KUKA KRL program: MyProgram_113().src

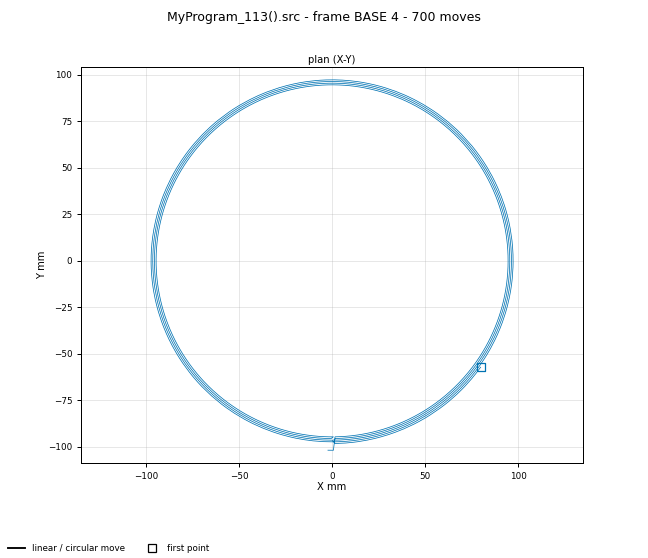
[picture p0: tool path of MyProgram_113().src in frame BASE 4, 700 of 700 moves have a stored position in this frame; points joined in program order, loops and branches not executed]
&ACCESS RVP
&REL 1
&PARAM TEMPLATE = C:\KRC\Roboter\Template\vorgabe
&PARAM EDITMASK = *
DEF MyProgram_113()
; ---- Setting reference (Base) ----
$BASE = BASE_DATA[4]

; --------------------------
; ---- Setting tool (TCP) ----
$TOOL = TOOL_DATA[3]
; --------------------------

$VEL.CP = VEL_APROX_PRINT
Startdeposition()
$VEL.CP = VEL_PRINT
LIN {X 79.7976,Y -57.1488,Z 98,A -40.8571,B 24.9367,C -1.8375,E1 25.1286,E2 126.2832} C_DIS
LIN {X 77.2204,Y -60.5867,Z 98,A -43.0229,B 24.9363,C -1.844,E1 25.125,E2 128.4234} C_DIS
LIN {X 74.8763,Y -63.4603,Z 98,A -45.4458,B 24.9373,C -1.8284,E1 25.1206,E2 130.8721} C_DIS
LIN {X 71.3027,Y -67.4509,Z 98,A -48.1343,B 24.9367,C -1.8374,E1 25.1156,E2 133.5274} C_DIS
LIN {X 69.3871,Y -69.4217,Z 98,A -49.9709,B 24.9376,C -1.8245,E1 25.1119,E2 135.3867} C_DIS
LIN {X 66.9172,Y -71.8046,Z 98,A -52.0394,B 24.9381,C -1.8172,E1 25.1077,E2 137.4638} C_DIS
LIN {X 62.9842,Y -75.2776,Z 98,A -54.7785,B 24.9377,C -1.8227,E1 25.102,E2 140.1792} C_DIS
LIN {X 60.5437,Y -77.2543,Z 98,A -56.7758,B 24.9384,C -1.8124,E1 25.0976,E2 142.1934} C_DIS
LIN {X 58.0242,Y -79.1632,Z 98,A -58.7964,B 24.9391,C -1.8018,E1 25.093,E2 144.2318} C_DIS
LIN {X 52.4588,Y -82.9577,Z 98,A -62.2953,B 24.9386,C -1.8106,E1 25.085,E2 147.6983} C_DIS
LIN {X 50.2118,Y -84.3355,Z 98,A -64.0193,B 24.9392,C -1.8007,E1 25.0808,E2 149.4404} C_DIS
LIN {X 46.9316,Y -86.2036,Z 98,A -66.5927,B 24.9404,C -1.7828,E1 25.0744,E2 152.0485} C_DIS
LIN {X 44.0309,Y -87.7219,Z 98,A -68.1285,B 24.9397,C -1.7938,E1 25.0707,E2 153.5542} C_DIS
LIN {X 38.5072,Y -90.2828,Z 98,A -71.4077,B 24.9394,C -1.7987,E1 25.0624,E2 156.8136} C_DIS
LIN {X 33.9539,Y -92.0916,Z 98,A -74.5314,B 24.9403,C -1.7848,E1 25.0542,E2 159.9633} C_DIS
LIN {X 30.3745,Y -93.3329,Z 98,A -76.7207,B 24.9404,C -1.7828,E1 25.0484,E2 162.1529} C_DIS
LIN {X 26.2417,Y -94.5794,Z 98,A -79.2585,B 24.9407,C -1.7793,E1 25.0416,E2 164.6947} C_DIS
LIN {X 22.9791,Y -95.4236,Z 98,A -81.814,B 24.9422,C -1.7557,E1 25.0345,E2 167.3025} C_DIS
LIN {X 18.9563,Y -96.3039,Z 98,A -83.7662,B 24.9413,C -1.7702,E1 25.0293,E2 169.218} C_DIS
LIN {X 13.978,Y -97.1507,Z 98,A -86.15,B 24.94,C -1.7888,E1 25.0228,E2 171.5551} C_DIS
LIN {X 11.5893,Y -97.4645,Z 98,A -88.6482,B 24.9427,C -1.7479,E1 25.0156,E2 174.1484} C_DIS
LIN {X 7.1702,Y -97.8893,Z 98,A -90.2748,B 24.9405,C -1.7818,E1 25.0113,E2 175.6938} C_DIS
LIN {X 1.7256,Y -98.1358,Z 98,A -93.4363,B 24.9405,C -1.7814,E1 25.0025,E2 178.8555} C_DIS
LIN {X 1.7256,Y -98.1358,Z 98,A -93.4363,B 24.9405,C -1.7814,E1 25.0025,E2 178.8555} C_DIS
Enddeposition()
LIN {X 0.7021,Y -97.2501,Z 98,A -94.9609,B 24.9417,C -1.7637,E1 24.9981,E2 180.4219} C_DIS
Startdeposition()
$VEL.CP = VEL_PRINT
LIN {X 3.3521,Y -97.1984,Z 98,A -91.5255,B 24.9371,C -1.832,E1 25.0082,E2 176.8251} C_DIS
LIN {X 7.9705,Y -96.9286,Z 98,A -88.6357,B 24.9366,C -1.8394,E1 25.0163,E2 173.9192} C_DIS
LIN {X 11.4013,Y -96.5849,Z 98,A -87.1457,B 24.9379,C -1.8205,E1 25.0203,E2 172.4751} C_DIS
LIN {X 14.7868,Y -96.1248,Z 98,A -85.2922,B 24.9382,C -1.8159,E1 25.0254,E2 170.6339} C_DIS
LIN {X 18.9278,Y -95.3974,Z 98,A -82.0938,B 24.9362,C -1.8449,E1 25.0343,E2 167.3706} C_DIS
LIN {X 22.4173,Y -94.6382,Z 98,A -80.5089,B 24.9374,C -1.8274,E1 25.0385,E2 165.8293} C_DIS
LIN {X 25.8034,Y -93.7711,Z 98,A -78.594,B 24.9376,C -1.8242,E1 25.0436,E2 163.9251} C_DIS
LIN {X 28.6619,Y -92.9362,Z 98,A -76.7124,B 24.9372,C -1.831,E1 25.0487,E2 162.0308} C_DIS
LIN {X 31.9858,Y -91.8454,Z 98,A -74.7403,B 24.9372,C -1.8302,E1 25.0539,E2 160.0644} C_DIS
LIN {X 36.6622,Y -90.0806,Z 98,A -71.8461,B 24.9371,C -1.8323,E1 25.0615,E2 157.1714} C_DIS
LIN {X 38.538,Y -89.2943,Z 98,A -69.8507,B 24.9348,C -1.8645,E1 25.0668,E2 155.1047} C_DIS
LIN {X 42.308,Y -87.5711,Z 98,A -68.0871,B 24.9364,C -1.8424,E1 25.0711,E2 153.398} C_DIS
LIN {X 44.7573,Y -86.3462,Z 98,A -66.3081,B 24.9357,C -1.8514,E1 25.0755,E2 151.6026} C_DIS
LIN {X 51.0632,Y -82.7737,Z 98,A -62.3793,B 24.9361,C -1.846,E1 25.085,E2 147.6983} C_DIS
LIN {X 55.4802,Y -79.8785,Z 98,A -58.6183,B 24.9339,C -1.8772,E1 25.0938,E2 143.8761} C_DIS
LIN {X 58.3576,Y -77.8012,Z 98,A -57.0633,B 24.9351,C -1.8609,E1 25.0972,E2 142.3654} C_DIS
LIN {X 61.0225,Y -75.7295,Z 98,A -55.3486,B 24.9355,C -1.8546,E1 25.1009,E2 140.6718} C_DIS
LIN {X 64.4955,Y -72.7957,Z 98,A -51.9466,B 24.9331,C -1.8888,E1 25.1082,E2 137.2025} C_DIS
LIN {X 66.9498,Y -70.5447,Z 98,A -50.4816,B 24.9342,C -1.8741,E1 25.1111,E2 135.7782} C_DIS
LIN {X 69.097,Y -68.4416,Z 98,A -48.7316,B 24.9339,C -1.8776,E1 25.1146,E2 134.0274} C_DIS
LIN {X 72.4346,Y -64.8989,Z 98,A -45.2556,B 24.9317,C -1.9087,E1 25.1213,E2 130.4932} C_DIS
LIN {X 74.9309,Y -62.0003,Z 98,A -43.6411,B 24.9331,C -1.8894,E1 25.1241,E2 128.9315} C_DIS
LIN {X 76.9346,Y -59.4956,Z 98,A -41.0568,B 24.9308,C -1.9218,E1 25.1286,E2 126.283} C_DIS
LIN {X 79.3962,Y -56.1696,Z 98,A -39.1586,B 24.9318,C -1.9072,E1 25.1316,E2 124.4285} C_DIS
LIN {X 81.8934,Y -52.4605,Z 98,A -36.5864,B 24.9315,C -1.9122,E1 25.1355,E2 121.8573} C_DIS
LIN {X 83.2034,Y -50.3573,Z 98,A -34.6449,B 24.9298,C -1.9354,E1 25.1384,E2 119.8709} C_DIS
LIN {X 85.1347,Y -47.0204,Z 98,A -33.2212,B 24.9317,C -1.9086,E1 25.1403,E2 118.518} C_DIS
LIN {X 87.4131,Y -42.6369,Z 98,A -29.992,B 24.9302,C -1.9297,E1 25.1444,E2 115.2561} C_DIS
LIN {X 88.8191,Y -39.6224,Z 98,A -28.2174,B 24.9302,C -1.9283,E1 25.1464,E2 113.4944} C_DIS
LIN {X 90.266,Y -36.2067,Z 98,A -25.8677,B 24.9293,C -1.9415,E1 25.149,E2 111.1265} C_DIS
LIN {X 91.5506,Y -32.8238,Z 98,A -23.7356,B 24.9288,C -1.9481,E1 25.151,E2 108.9907} C_DIS
LIN {X 93.2043,Y -27.7776,Z 98,A -20.6688,B 24.9283,C -1.9555,E1 25.1536,E2 105.924} C_DIS
LIN {X 94.208,Y -24.1556,Z 98,A -18.5095,B 24.9279,C -1.9603,E1 25.1552,E2 103.7657} C_DIS
LIN {X 95.2371,Y -19.7115,Z 98,A -16.2285,B 24.9285,C -1.9529,E1 25.1566,E2 101.5155} C_DIS
LIN {X 95.9344,Y -15.9756,Z 98,A -13.6784,B 24.9271,C -1.9723,E1 25.1578,E2 98.9345} C_DIS
LIN {X 96.4194,Y -12.7275,Z 98,A -11.7354,B 24.9266,C -1.9788,E1 25.1586,E2 96.9876} C_DIS
LIN {X 96.7838,Y -9.5822,Z 98,A -9.6481,B 24.9255,C -1.9936,E1 25.1592,E2 94.8777} C_DIS
LIN {X 97.1972,Y -3.3908,Z 98,A -6.1803,B 24.9252,C -1.998,E1 25.1597,E2 91.4203} C_DIS
LIN {X 97.2518,Y -0.8973,Z 98,A -4.0584,B 24.9228,C -2.0287,E1 25.1597,E2 89.2385} C_DIS
LIN {X 97.1951,Y 3.4602,Z 98,A -2.3961,B 24.9249,C -2.0009,E1 25.1597,E2 87.6515} C_DIS
LIN {X 96.9672,Y 7.4872,Z 98,A 0.1195,B 24.9239,C -2.014,E1 25.1592,E2 85.12} C_DIS
LIN {X 96.6458,Y 10.8814,Z 98,A 2.1602,B 24.9234,C -2.0217,E1 25.1586,E2 83.0734} C_DIS
LIN {X 95.684,Y 17.4137,Z 98,A 6.0714,B 24.9224,C -2.0347,E1 25.1569,E2 79.1543} C_DIS
LIN {X 94.9676,Y 20.9723,Z 98,A 8.0982,B 24.9222,C -2.0369,E1 25.1557,E2 77.1341} C_DIS
LIN {X 94.1017,Y 24.5689,Z 98,A 10.2032,B 24.9219,C -2.0407,E1 25.1543,E2 75.0324} C_DIS
LIN {X 93.2925,Y 27.4805,Z 98,A 12.0287,B 24.9214,C -2.0479,E1 25.1529,E2 73.2003} C_DIS
LIN {X 92.4694,Y 30.1344,Z 98,A 14.4718,B 24.9185,C -2.0846,E1 25.1507,E2 70.6845} C_DIS
LIN {X 90.9388,Y 34.4784,Z 98,A 16.3375,B 24.9205,C -2.0592,E1 25.149,E2 68.8892} C_DIS
LIN {X 89.01,Y 39.1915,Z 98,A 19.9629,B 24.9179,C -2.0923,E1 25.145,E2 65.2054} C_DIS
LIN {X 87.3478,Y 42.7693,Z 98,A 21.6868,B 24.9192,C -2.0753,E1 25.1429,E2 63.531} C_DIS
LIN {X 85.9471,Y 45.5167,Z 98,A 24.5151,B 24.9157,C -2.12,E1 25.1391,E2 60.612} C_DIS
LIN {X 83.2177,Y 50.3337,Z 98,A 27.2311,B 24.9167,C -2.1072,E1 25.1352,E2 57.9401} C_DIS
LIN {X 81.3082,Y 53.3634,Z 98,A 29.2555,B 24.9166,C -2.1093,E1 25.1322,E2 55.9209} C_DIS
LIN {X 79.4218,Y 56.1337,Z 98,A 30.8335,B 24.9174,C -2.0988,E1 25.1297,E2 54.3753} C_DIS
LIN {X 77.2022,Y 59.1483,Z 98,A 33.4101,B 24.9158,C -2.1186,E1 25.1253,E2 51.7642} C_DIS
LIN {X 75.1203,Y 61.7724,Z 98,A 35.1259,B 24.9162,C -2.1133,E1 25.1223,E2 50.069} C_DIS
LIN {X 69.4071,Y 68.1276,Z 98,A 39.9538,B 24.916,C -2.1165,E1 25.1132,E2 45.2548} C_DIS
LIN {X 67.1097,Y 70.3932,Z 98,A 42.2478,B 24.9145,C -2.1355,E1 25.1085,E2 42.9253} C_DIS
LIN {X 62.2387,Y 74.7328,Z 98,A 45.8912,B 24.9145,C -2.1354,E1 25.1008,E2 39.2965} C_DIS
LIN {X 56.8744,Y 78.8933,Z 98,A 49.6994,B 24.9145,C -2.1352,E1 25.0924,E2 35.5026} C_DIS
LIN {X 53.8448,Y 80.9908,Z 98,A 52.9079,B 24.911,C -2.1781,E1 25.0847,E2 32.2033} C_DIS
LIN {X 48.9624,Y 84.0336,Z 98,A 55.057,B 24.9144,C -2.1362,E1 25.0798,E2 30.16} C_DIS
LIN {X 44.2162,Y 86.6231,Z 98,A 58.4066,B 24.9136,C -2.1466,E1 25.0715,E2 26.7953} C_DIS
LIN {X 40.9897,Y 88.1956,Z 98,A 60.4692,B 24.9136,C -2.1472,E1 25.0663,E2 24.7366} C_DIS
LIN {X 38.9606,Y 89.1106,Z 98,A 62.7877,B 24.9103,C -2.1862,E1 25.0602,E2 22.3313} C_DIS
LIN {X 33.9331,Y 91.1453,Z 98,A 64.9612,B 24.9132,C -2.1512,E1 25.0547,E2 20.2454} C_DIS
LIN {X 28.6134,Y 92.9513,Z 98,A 68.0623,B 24.9136,C -2.1463,E1 25.0466,E2 17.1619} C_DIS
LIN {X 25.915,Y 93.7406,Z 98,A 69.9785,B 24.9127,C -2.1569,E1 25.0414,E2 15.2237} C_DIS
LIN {X 22.9884,Y 94.4995,Z 98,A 71.6259,B 24.913,C -2.1531,E1 25.0369,E2 13.5878} C_DIS
LIN {X 19.7066,Y 95.2381,Z 98,A 73.6718,B 24.9128,C -2.1564,E1 25.0313,E2 11.5368} C_DIS
LIN {X 16.4675,Y 95.8522,Z 98,A 75.666,B 24.9126,C -2.159,E1 25.0258,E2 9.5386} C_DIS
LIN {X 13.9554,Y 96.2494,Z 98,A 77.9138,B 24.9103,C -2.1866,E1 25.0195,E2 7.2272} C_DIS
LIN {X 9.3981,Y 96.8014,Z 98,A 79.9182,B 24.9124,C -2.1616,E1 25.0141,E2 5.2835} C_DIS
LIN {X 5.6176,Y 97.0934,Z 98,A 81.9493,B 24.9129,C -2.1544,E1 25.0084,E2 3.2704} C_DIS
LIN {X 1.3581,Y 97.247,Z 98,A 84.4198,B 24.9131,C -2.1527,E1 25.0016,E2 0.8045} C_DIS
LIN {X -3.1957,Y 97.2032,Z 98,A 87.2707,B 24.9127,C -2.158,E1 24.9936,E2 -2.0591} C_DIS
LIN {X -6.5423,Y 97.0352,Z 98,A 89.0987,B 24.9131,C -2.1521,E1 24.9885,E2 -3.8736} C_DIS
LIN {X -8.6993,Y 96.8659,Z 98,A 90.8129,B 24.9119,C -2.167,E1 24.9836,E2 -5.6241} C_DIS
LIN {X -14.1209,Y 96.2259,Z 98,A 93.7478,B 24.9129,C -2.1551,E1 24.9756,E2 -8.5328} C_DIS
LIN {X -17.3852,Y 95.6892,Z 98,A 95.5906,B 24.9133,C -2.1499,E1 24.9705,E2 -10.3653} C_DIS
LIN {X -20.594,Y 95.0502,Z 98,A 97.6154,B 24.9132,C -2.1517,E1 24.965,E2 -12.3966} C_DIS
LIN {X -24.4571,Y 94.1305,Z 98,A 100.7061,B 24.9112,C -2.1757,E1 24.9565,E2 -15.5489} C_DIS
LIN {X -28.6765,Y 92.9317,Z 98,A 102.5615,B 24.9135,C -2.1474,E1 24.9517,E2 -17.3401} C_DIS
LIN {X -34.996,Y 90.7419,Z 98,A 106.4035,B 24.9142,C -2.139,E1 24.9416,E2 -21.1696} C_DIS
LIN {X -39.6014,Y 88.8282,Z 98,A 109.857,B 24.9131,C -2.1524,E1 24.9326,E2 -24.6633} C_DIS
LIN {X -44.1812,Y 86.641,Z 98,A 112.429,B 24.9146,C -2.1333,E1 24.9263,E2 -27.1965} C_DIS
LIN {X -50.0589,Y 83.3847,Z 98,A 116.4561,B 24.915,C -2.1286,E1 24.9165,E2 -31.2242} C_DIS
LIN {X -52.8436,Y 81.6475,Z 98,A 118.4417,B 24.9152,C -2.1268,E1 24.9118,E2 -33.2118} C_DIS
LIN {X -55.4064,Y 79.9298,Z 98,A 120.486,B 24.9148,C -2.1308,E1 24.9071,E2 -35.2727} C_DIS
LIN {X -60.9712,Y 75.7711,Z 98,A 124.3317,B 24.9162,C -2.1138,E1 24.8986,E2 -39.0918} C_DIS
LIN {X -62.9622,Y 74.1243,Z 98,A 126.2604,B 24.9154,C -2.1241,E1 24.8944,E2 -41.0525} C_DIS
LIN {X -65.4196,Y 71.966,Z 98,A 127.5675,B 24.9174,C -2.0989,E1 24.8918,E2 -42.3048} C_DIS
LIN {X -69.6493,Y 67.8814,Z 98,A 131.1261,B 24.9178,C -2.0937,E1 24.8847,E2 -45.8659} C_DIS
LIN {X -73.917,Y 63.2055,Z 98,A 135.7169,B 24.9163,C -2.113,E1 24.8761,E2 -50.5232} C_DIS
LIN {X -76.658,Y 59.854,Z 98,A 137.6654,B 24.9184,C -2.0861,E1 24.8728,E2 -52.4168} C_DIS
LIN {X -78.4849,Y 57.4348,Z 98,A 140.0476,B 24.9172,C -2.1011,E1 24.8688,E2 -54.8464} C_DIS
LIN {X -80.8866,Y 54.0016,Z 98,A 142.1963,B 24.9186,C -2.0836,E1 24.8655,E2 -56.964} C_DIS
LIN {X -83.2691,Y 50.2492,Z 98,A 144.5739,B 24.9198,C -2.0682,E1 24.8621,E2 -59.317} C_DIS
LIN {X -85.0659,Y 47.1436,Z 98,A 146.7028,B 24.9202,C -2.0626,E1 24.8591,E2 -61.4437} C_DIS
LIN {X -86.7141,Y 44.038,Z 98,A 148.614,B 24.9211,C -2.0513,E1 24.8567,E2 -63.338} C_DIS
LIN {X -89.1122,Y 38.957,Z 98,A 152.0493,B 24.9215,C -2.0454,E1 24.8527,E2 -66.7781} C_DIS
LIN {X -90.7245,Y 35.0428,Z 98,A 154.6329,B 24.9219,C -2.0407,E1 24.85,E2 -69.3648} C_DIS
LIN {X -91.7647,Y 32.216,Z 98,A 157.0901,B 24.9206,C -2.0577,E1 24.8477,E2 -71.8765} C_DIS
LIN {X -93.1472,Y 27.9702,Z 98,A 158.7019,B 24.9238,C -2.016,E1 24.8464,E2 -73.3981} C_DIS
LIN {X -93.962,Y 25.0964,Z 98,A 161.2031,B 24.9224,C -2.0347,E1 24.8445,E2 -75.9584} C_DIS
LIN {X -94.7586,Y 21.8958,Z 98,A 162.5158,B 24.9244,C -2.0079,E1 24.8437,E2 -77.2149} C_DIS
LIN {X -95.7485,Y 17.0551,Z 98,A 165.8704,B 24.924,C -2.013,E1 24.8419,E2 -80.6016} C_DIS
LIN {X -96.3963,Y 12.9055,Z 98,A 168.184,B 24.925,C -1.9998,E1 24.841,E2 -82.8976} C_DIS
LIN {X -96.8017,Y 9.3948,Z 98,A 170.2948,B 24.9254,C -1.9941,E1 24.8404,E2 -85.0073} C_DIS
LIN {X -97.0833,Y 5.8008,Z 98,A 172.4018,B 24.926,C -1.9867,E1 24.84,E2 -87.1093} C_DIS
LIN {X -97.2182,Y 2.7075,Z 98,A 174.3229,B 24.9262,C -1.984,E1 24.8398,E2 -89.0355} C_DIS
LIN {X -97.2492,Y -1.2353,Z 98,A 176.5717,B 24.9269,C -1.9741,E1 24.8398,E2 -91.2742} C_DIS
LIN {X -97.1784,Y -3.8816,Z 98,A 178.1999,B 24.9271,C -1.9714,E1 24.84,E2 -92.9058} C_DIS
LIN {X -96.9749,Y -7.3909,Z 98,A -179.7635,B 24.9277,C -1.9636,E1 24.8404,E2 -94.9361} C_DIS
LIN {X -96.6498,Y -10.8471,Z 98,A -177.7048,B 24.9282,C -1.9576,E1 24.841,E2 -96.9927} C_DIS
LIN {X -96.2055,Y -14.2638,Z 98,A -175.8318,B 24.929,C -1.946,E1 24.8417,E2 -98.8494} C_DIS
LIN {X -95.8403,Y -16.5341,Z 98,A -173.7061,B 24.9274,C -1.9672,E1 24.8427,E2 -101.0382} C_DIS
LIN {X -95.0898,Y -20.4121,Z 98,A -171.9685,B 24.9294,C -1.9405,E1 24.8437,E2 -102.7223} C_DIS
LIN {X -94.3321,Y -23.6726,Z 98,A -169.4325,B 24.9285,C -1.9531,E1 24.8454,E2 -105.3031} C_DIS
LIN {X -93.3638,Y -27.2383,Z 98,A -167.9504,B 24.9306,C -1.9235,E1 24.8465,E2 -106.7233} C_DIS
LIN {X -91.7681,Y -32.2062,Z 98,A -164.7711,B 24.931,C -1.9178,E1 24.8493,E2 -109.9072} C_DIS
LIN {X -90.5811,Y -35.4079,Z 98,A -162.6045,B 24.9311,C -1.917,E1 24.8515,E2 -112.0841} C_DIS
LIN {X -89.0286,Y -39.1488,Z 98,A -160.2193,B 24.9316,C -1.9101,E1 24.8541,E2 -114.4661} C_DIS
LIN {X -87.6653,Y -42.112,Z 98,A -158.3747,B 24.9322,C -1.9022,E1 24.8563,E2 -116.3017} C_DIS
LIN {X -85.9482,Y -45.5146,Z 98,A -155.8134,B 24.9319,C -1.9065,E1 24.8596,E2 -118.8871} C_DIS
LIN {X -83.7352,Y -49.4677,Z 98,A -153.6079,B 24.9335,C -1.8839,E1 24.8626,E2 -121.0502} C_DIS
LIN {X -81.9113,Y -52.4326,Z 98,A -151.4265,B 24.9335,C -1.8829,E1 24.8658,E2 -123.2403} C_DIS
LIN {X -80.1435,Y -55.0991,Z 98,A -149.6354,B 24.9341,C -1.875,E1 24.8686,E2 -125.0213} C_DIS
LIN {X -76.7363,Y -59.7529,Z 98,A -145.9637,B 24.9341,C -1.8758,E1 24.8748,E2 -128.7127} C_DIS
LIN {X -74.4696,Y -62.5554,Z 98,A -144.1062,B 24.935,C -1.8619,E1 24.878,E2 -130.5456} C_DIS
LIN {X -72.1623,Y -65.2006,Z 98,A -141.6555,B 24.9344,C -1.8702,E1 24.8826,E2 -133.0271} C_DIS
LIN {X -69.846,Y -67.6774,Z 98,A -139.4169,B 24.9342,C -1.874,E1 24.887,E2 -135.2846} C_DIS
LIN {X -64.7417,Y -72.5752,Z 98,A -135.5848,B 24.9356,C -1.8541,E1 24.8947,E2 -139.0848} C_DIS
LIN {X -59.452,Y -76.9682,Z 98,A -131.5912,B 24.9362,C -1.8445,E1 24.9034,E2 -143.0707} C_DIS
LIN {X -56.6774,Y -79.0339,Z 98,A -128.5574,B 24.934,C -1.8757,E1 24.9104,E2 -146.1893} C_DIS
LIN {X -52.3814,Y -81.9442,Z 98,A -126.3909,B 24.9366,C -1.8398,E1 24.9153,E2 -148.2773} C_DIS
LIN {X -47.0051,Y -85.1432,Z 98,A -122.7464,B 24.937,C -1.833,E1 24.9241,E2 -151.9167} C_DIS
LIN {X -43.9173,Y -86.7758,Z 98,A -120.6954,B 24.9372,C -1.8302,E1 24.9292,E2 -153.9665} C_DIS
LIN {X -41.8772,Y -87.7781,Z 98,A -118.3957,B 24.935,C -1.8626,E1 24.9352,E2 -156.3491} C_DIS
LIN {X -37.1314,Y -89.8896,Z 98,A -116.2478,B 24.9374,C -1.827,E1 24.9405,E2 -158.4173} C_DIS
LIN {X -31.8211,Y -91.9033,Z 98,A -113.092,B 24.9381,C -1.8172,E1 24.9487,E2 -161.5563} C_DIS
LIN {X -29.1166,Y -92.7952,Z 98,A -111.2627,B 24.9378,C -1.8213,E1 24.9536,E2 -163.3986} C_DIS
LIN {X -26.8573,Y -93.4743,Z 98,A -109.1966,B 24.9362,C -1.8446,E1 24.9594,E2 -165.5235} C_DIS
LIN {X -22.9393,Y -94.5115,Z 98,A -107.4573,B 24.9379,C -1.82,E1 24.9639,E2 -167.2067} C_DIS
LIN {X -19.4891,Y -95.2828,Z 98,A -105.3266,B 24.9379,C -1.8207,E1 24.9697,E2 -169.3417} C_DIS
LIN {X -14.9197,Y -96.1043,Z 98,A -102.3002,B 24.9372,C -1.8305,E1 24.9781,E2 -172.3941} C_DIS
LIN {X -10.2422,Y -96.7147,Z 98,A -99.8486,B 24.938,C -1.8181,E1 24.9849,E2 -174.8181} C_DIS
LIN {X -4.8097,Y -97.1381,Z 98,A -96.7684,B 24.9384,C -1.8134,E1 24.9934,E2 -177.8881} C_DIS
LIN {X 0.7021,Y -97.2501,Z 98,A -94.9572,B 24.9418,C -1.7621,E1 24.9982,E2 -179.5782} C_DIS
Enddeposition()
LIN {X 0.7021,Y -97.2501,Z 98,A -94.9572,B 24.9418,C -1.7621,E1 24.9982,E2 -179.5782} C_DIS
Startdeposition()
$VEL.CP = VEL_PRINT
LIN {X 0.1199,Y -96.3611,Z 98,A -95.1066,B 24.9403,C -1.7848,E1 24.9979,E2 -179.4825} C_DIS
LIN {X -4.7533,Y -96.2443,Z 98,A -97.7417,B 24.9397,C -1.7938,E1 24.9906,E2 -176.8682} C_DIS
LIN {X -8.6799,Y -95.9684,Z 98,A -99.885,B 24.9392,C -1.8009,E1 24.9846,E2 -174.7407} C_DIS
LIN {X -11.7051,Y -95.6477,Z 98,A -101.5908,B 24.939,C -1.8047,E1 24.9799,E2 -173.0429} C_DIS
LIN {X -14.4371,Y -95.2728,Z 98,A -103.4664,B 24.9395,C -1.7968,E1 24.9747,E2 -171.1471} C_DIS
LIN {X -18.3264,Y -94.6013,Z 98,A -105.6647,B 24.9391,C -1.8028,E1 24.9687,E2 -168.9608} C_DIS
LIN {X -21.3205,Y -93.9725,Z 98,A -107.5616,B 24.9392,C -1.801,E1 24.9635,E2 -167.0571} C_DIS
LIN {X -26.2275,Y -92.722,Z 98,A -110.4859,B 24.9389,C -1.8058,E1 24.9556,E2 -164.1398} C_DIS
LIN {X -29.7956,Y -91.6378,Z 98,A -112.7098,B 24.9388,C -1.8072,E1 24.9497,E2 -161.9154} C_DIS
LIN {X -33.227,Y -90.4503,Z 98,A -115.0181,B 24.939,C -1.8039,E1 24.9436,E2 -159.5947} C_DIS
LIN {X -36.5664,Y -89.1528,Z 98,A -116.9313,B 24.9384,C -1.8134,E1 24.9387,E2 -157.7} C_DIS
LIN {X -40.9689,Y -87.2176,Z 98,A -120.0125,B 24.9387,C -1.809,E1 24.9308,E2 -154.6008} C_DIS
LIN {X -44.0738,Y -85.6902,Z 98,A -121.9763,B 24.9383,C -1.8147,E1 24.9259,E2 -152.6454} C_DIS
LIN {X -46.6259,Y -84.3293,Z 98,A -124.1126,B 24.9391,C -1.803,E1 24.9206,E2 -150.4751} C_DIS
LIN {X -50.8414,Y -81.8563,Z 98,A -126.6574,B 24.938,C -1.8194,E1 24.9146,E2 -147.9614} C_DIS
LIN {X -53.0392,Y -80.4493,Z 98,A -128.7257,B 24.939,C -1.8046,E1 24.9097,E2 -145.8511} C_DIS
LIN {X -55.9684,Y -78.4397,Z 98,A -130.3415,B 24.9376,C -1.8246,E1 24.9061,E2 -144.2776} C_DIS
LIN {X -58.6788,Y -76.4335,Z 98,A -132.7683,B 24.9383,C -1.8141,E1 24.9006,E2 -141.817} C_DIS
LIN {X -61.2432,Y -74.3957,Z 98,A -134.3282,B 24.9372,C -1.8306,E1 24.8973,E2 -140.2903} C_DIS
LIN {X -63.8595,Y -72.1631,Z 98,A -136.2165,B 24.9366,C -1.8397,E1 24.8933,E2 -138.4165} C_DIS
LIN {X -66.996,Y -69.259,Z 98,A -139.3854,B 24.9376,C -1.8243,E1 24.8868,E2 -135.1977} C_DIS
LIN {X -69.406,Y -66.8435,Z 98,A -140.4596,B 24.9351,C -1.8601,E1 24.8849,E2 -134.2042} C_DIS
LIN {X -72.7402,Y -63.1995,Z 98,A -143.9622,B 24.936,C -1.8479,E1 24.8782,E2 -130.657} C_DIS
LIN {X -75.0181,Y -60.4781,Z 98,A -146.0938,B 24.9357,C -1.8522,E1 24.8744,E2 -128.5257} C_DIS
LIN {X -76.9771,Y -57.9636,Z 98,A -148.3432,B 24.9362,C -1.8453,E1 24.8706,E2 -126.2491} C_DIS
LIN {X -78.8902,Y -55.3331,Z 98,A -149.8767,B 24.9349,C -1.8631,E1 24.8682,E2 -124.7505} C_DIS
LIN {X -80.6765,Y -52.6946,Z 98,A -151.6024,B 24.9342,C -1.8734,E1 24.8655,E2 -123.0408} C_DIS
LIN {X -82.0591,Y -50.5159,Z 98,A -153.2874,B 24.9342,C -1.8725,E1 24.863,E2 -121.345} C_DIS
LIN {X -83.7685,Y -47.6265,Z 98,A -155.1345,B 24.9336,C -1.8826,E1 24.8604,E2 -119.5125} C_DIS
LIN {X -85.7944,Y -43.87,Z 98,A -157.7317,B 24.9332,C -1.8876,E1 24.857,E2 -116.9135} C_DIS
LIN {X -87.2479,Y -40.9038,Z 98,A -159.7968,B 24.933,C -1.8899,E1 24.8545,E2 -114.8426} C_DIS
LIN {X -88.4821,Y -38.1616,Z 98,A -161.5183,B 24.9325,C -1.8971,E1 24.8526,E2 -113.1288} C_DIS
LIN {X -89.6391,Y -35.3567,Z 98,A -163.4277,B 24.9324,C -1.899,E1 24.8506,E2 -111.2132} C_DIS
LIN {X -90.816,Y -32.2152,Z 98,A -165.28,B 24.9317,C -1.9094,E1 24.8488,E2 -109.3753} C_DIS
LIN {X -92.039,Y -28.5318,Z 98,A -167.3952,B 24.9307,C -1.9225,E1 24.847,E2 -107.2792} C_DIS
LIN {X -93.1328,Y -24.7318,Z 98,A -170.3875,B 24.9317,C -1.9091,E1 24.8447,E2 -104.2376} C_DIS
LIN {X -93.9973,Y -21.2132,Z 98,A -172.4925,B 24.9311,C -1.9173,E1 24.8433,E2 -102.1398} C_DIS
LIN {X -95.2551,Y -14.5517,Z 98,A -176.3378,B 24.9297,C -1.9358,E1 24.8415,E2 -98.3158} C_DIS
LIN {X -95.6795,Y -11.4341,Z 98,A -178.2904,B 24.9295,C -1.9391,E1 24.8408,E2 -96.3595} C_DIS
LIN {X -96.0348,Y -7.9137,Z 98,A 179.6587,B 24.9289,C -1.9474,E1 24.8402,E2 -94.3162} C_DIS
LIN {X -96.2637,Y -4.3109,Z 98,A 177.3664,B 24.9287,C -1.9497,E1 24.8399,E2 -92.0154} C_DIS
LIN {X -96.358,Y -0.6033,Z 98,A 175.2696,B 24.928,C -1.9602,E1 24.8398,E2 -89.9311} C_DIS
LIN {X -96.3089,Y 3.1422,Z 98,A 172.9059,B 24.9278,C -1.963,E1 24.8399,E2 -87.56} C_DIS
LIN {X -96.1317,Y 6.6299,Z 98,A 170.8376,B 24.9272,C -1.97,E1 24.8403,E2 -85.4958} C_DIS
LIN {X -95.8437,Y 9.9621,Z 98,A 168.9084,B 24.9266,C -1.9783,E1 24.8408,E2 -83.5748} C_DIS
LIN {X -95.4593,Y 13.1507,Z 98,A 166.6895,B 24.9269,C -1.9746,E1 24.8416,E2 -81.3339} C_DIS
LIN {X -94.2571,Y 20.0277,Z 98,A 162.746,B 24.9254,C -1.9944,E1 24.8436,E2 -77.4144} C_DIS
LIN {X -92.5657,Y 26.779,Z 98,A 158.5742,B 24.9245,C -2.0065,E1 24.8466,E2 -73.2469} C_DIS
LIN {X -91.1897,Y 31.1421,Z 98,A 155.8199,B 24.924,C -2.0139,E1 24.8489,E2 -70.4945} C_DIS
LIN {X -89.9518,Y 34.5561,Z 98,A 153.6989,B 24.9234,C -2.0217,E1 24.851,E2 -68.3803} C_DIS
LIN {X -88.4866,Y 38.1514,Z 98,A 151.5623,B 24.9224,C -2.0342,E1 24.8532,E2 -66.2617} C_DIS
LIN {X -86.3693,Y 42.727,Z 98,A 148.3616,B 24.9222,C -2.0367,E1 24.8571,E2 -63.0495} C_DIS
LIN {X -84.8071,Y 45.75,Z 98,A 146.4154,B 24.9216,C -2.0451,E1 24.8596,E2 -61.113} C_DIS
LIN {X -83.3828,Y 48.2977,Z 98,A 144.5923,B 24.9214,C -2.0473,E1 24.8621,E2 -59.2857} C_DIS
LIN {X -81.4154,Y 51.5473,Z 98,A 142.2079,B 24.9212,C -2.0497,E1 24.8656,E2 -56.8947} C_DIS
LIN {X -78.6881,Y 55.6202,Z 98,A 139.2918,B 24.9206,C -2.0577,E1 24.8702,E2 -53.9834} C_DIS
LIN {X -76.5021,Y 58.5898,Z 98,A 137.1728,B 24.92,C -2.066,E1 24.8737,E2 -51.8738} C_DIS
LIN {X -73.7676,Y 61.9981,Z 98,A 133.9594,B 24.921,C -2.0531,E1 24.8795,E2 -48.6149} C_DIS
LIN {X -71.263,Y 64.8613,Z 98,A 132.2458,B 24.9192,C -2.0763,E1 24.8826,E2 -46.949} C_DIS
LIN {X -68.7981,Y 67.4699,Z 98,A 130.3989,B 24.918,C -2.0909,E1 24.8862,E2 -45.1287} C_DIS
LIN {X -66.1036,Y 70.1112,Z 98,A 127.5515,B 24.9191,C -2.0767,E1 24.892,E2 -42.2357} C_DIS
LIN {X -62.6758,Y 73.1919,Z 98,A 125.119,B 24.9179,C -2.0928,E1 24.897,E2 -39.8321} C_DIS
LIN {X -59.5459,Y 75.7602,Z 98,A 122.4464,B 24.9181,C -2.0894,E1 24.9029,E2 -37.1415} C_DIS
LIN {X -55.523,Y 78.7573,Z 98,A 119.6423,B 24.9172,C -2.1014,E1 24.9092,E2 -34.3559} C_DIS
LIN {X -52.8282,Y 80.5884,Z 98,A 117.7519,B 24.9168,C -2.1067,E1 24.9135,E2 -32.4718} C_DIS
LIN {X -49.8534,Y 82.4617,Z 98,A 115.7549,B 24.9162,C -2.1136,E1 24.9183,E2 -30.4852} C_DIS
LIN {X -45.5705,Y 84.9044,Z 98,A 112.667,B 24.9162,C -2.1136,E1 24.9258,E2 -27.3881} C_DIS
LIN {X -43.415,Y 86.0269,Z 98,A 110.8591,B 24.917,C -2.1039,E1 24.9304,E2 -25.5524} C_DIS
LIN {X -37.9993,Y 88.5529,Z 98,A 107.6153,B 24.9158,C -2.1195,E1 24.9386,E2 -22.3378} C_DIS
LIN {X -34.9668,Y 89.7923,Z 98,A 105.1035,B 24.917,C -2.1034,E1 24.9452,E2 -19.7825} C_DIS
LIN {X -31.1829,Y 91.1759,Z 98,A 103.2259,B 24.9154,C -2.1236,E1 24.95,E2 -17.9491} C_DIS
LIN {X -23.7663,Y 93.3834,Z 98,A 98.723,B 24.9148,C -2.1319,E1 24.9621,E2 -13.4586} C_DIS
LIN {X -20.8637,Y 94.0748,Z 98,A 96.8509,B 24.9148,C -2.1302,E1 24.9672,E2 -11.5799} C_DIS
LIN {X -16.9287,Y 94.8614,Z 98,A 94.6239,B 24.9143,C -2.1375,E1 24.9733,E2 -9.368} C_DIS
LIN {X -13.3199,Y 95.4352,Z 98,A 91.7022,B 24.9162,C -2.1135,E1 24.9815,E2 -6.3868} C_DIS
LIN {X -9.1762,Y 95.9226,Z 98,A 89.9038,B 24.9143,C -2.138,E1 24.9864,E2 -4.6457} C_DIS
LIN {X -5.6901,Y 96.1926,Z 98,A 87.7615,B 24.9143,C -2.1367,E1 24.9923,E2 -2.4994} C_DIS
LIN {X -2.4083,Y 96.3315,Z 98,A 85.5968,B 24.9149,C -2.1299,E1 24.9984,E2 -0.3185} C_DIS
LIN {X 1.423,Y 96.3501,Z 98,A 83.4636,B 24.9145,C -2.1353,E1 25.0043,E2 1.8017} C_DIS
LIN {X 5.1973,Y 96.2198,Z 98,A 81.3372,B 24.9141,C -2.1396,E1 25.0102,E2 3.9174} C_DIS
LIN {X 8.6466,Y 95.9715,Z 98,A 79.4554,B 24.9137,C -2.1456,E1 25.0154,E2 5.784} C_DIS
LIN {X 13.0821,Y 95.469,Z 98,A 76.5969,B 24.9143,C -2.1379,E1 25.0234,E2 8.6586} C_DIS
LIN {X 16.2772,Y 94.9761,Z 98,A 74.6662,B 24.9143,C -2.137,E1 25.0287,E2 10.5895} C_DIS
LIN {X 19.5929,Y 94.3473,Z 98,A 72.6278,B 24.9145,C -2.135,E1 25.0343,E2 12.6303} C_DIS
LIN {X 23.0689,Y 93.5582,Z 98,A 70.6899,B 24.9141,C -2.1403,E1 25.0395,E2 14.5529} C_DIS
LIN {X 26.6973,Y 92.5889,Z 98,A 68.3878,B 24.9144,C -2.1363,E1 25.0458,E2 16.8606} C_DIS
LIN {X 30.3385,Y 91.4603,Z 98,A 66.1373,B 24.9145,C -2.1351,E1 25.0517,E2 19.1098} C_DIS
LIN {X 33.1593,Y 90.475,Z 98,A 64.4238,B 24.9145,C -2.1358,E1 25.0562,E2 20.8182} C_DIS
LIN {X 37.9111,Y 88.5905,Z 98,A 61.2526,B 24.9151,C -2.1279,E1 25.0645,E2 24.0008} C_DIS
LIN {X 40.9631,Y 87.2203,Z 98,A 59.274,B 24.9152,C -2.126,E1 25.0695,E2 25.979} C_DIS
LIN {X 43.9946,Y 85.7307,Z 98,A 56.7639,B 24.9169,C -2.1053,E1 25.0758,E2 28.531} C_DIS
LIN {X 47.2164,Y 83.9996,Z 98,A 55.0613,B 24.9158,C -2.1194,E1 25.0799,E2 30.1954} C_DIS
LIN {X 49.601,Y 82.6151,Z 98,A 52.9234,B 24.9174,C -2.0988,E1 25.0851,E2 32.3753} C_DIS
LIN {X 52.7695,Y 80.6271,Z 98,A 51.2439,B 24.9161,C -2.1151,E1 25.089,E2 34.0108} C_DIS
LIN {X 55.7823,Y 78.5725,Z 98,A 49.4572,B 24.9153,C -2.1256,E1 25.093,E2 35.7668} C_DIS
LIN {X 60.3774,Y 75.0997,Z 98,A 45.6926,B 24.9168,C -2.1068,E1 25.1014,E2 39.5618} C_DIS
LIN {X 63.6394,Y 72.3546,Z 98,A 42.3833,B 24.9194,C -2.0735,E1 25.1085,E2 42.9371} C_DIS
LIN {X 67.0559,Y 69.2013,Z 98,A 40.431,B 24.9175,C -2.0976,E1 25.1123,E2 44.8241} C_DIS
LIN {X 71.3814,Y 64.7317,Z 98,A 36.708,B 24.9182,C -2.0886,E1 25.1195,E2 48.5523} C_DIS
LIN {X 73.6623,Y 62.1236,Z 98,A 34.0678,B 24.9202,C -2.0622,E1 25.1244,E2 51.2428} C_DIS
LIN {X 76.1553,Y 59.0398,Z 98,A 32.3837,B 24.9187,C -2.0817,E1 25.1272,E2 52.873} C_DIS
LIN {X 78.0809,Y 56.4707,Z 98,A 30.5886,B 24.9187,C -2.0813,E1 25.1301,E2 54.6605} C_DIS
LIN {X 81.3685,Y 51.6205,Z 98,A 26.9216,B 24.92,C -2.0654,E1 25.1359,E2 58.3467} C_DIS
LIN {X 83.2152,Y 48.5874,Z 98,A 24.3637,B 24.9217,C -2.043,E1 25.1395,E2 60.9444} C_DIS
LIN {X 84.9913,Y 45.4098,Z 98,A 22.7102,B 24.9207,C -2.0563,E1 25.1417,E2 62.5577} C_DIS
LIN {X 86.4515,Y 42.5611,Z 98,A 21.0685,B 24.9203,C -2.061,E1 25.1437,E2 64.1797} C_DIS
LIN {X 88.7818,Y 37.4572,Z 98,A 17.5354,B 24.9217,C -2.044,E1 25.1478,E2 67.7338} C_DIS
LIN {X 90.017,Y 34.384,Z 98,A 15.472,B 24.9224,C -2.0347,E1 25.1499,E2 69.8077} C_DIS
LIN {X 91.7302,Y 29.51,Z 98,A 12.5184,B 24.9227,C -2.03,E1 25.1526,E2 72.7557} C_DIS
LIN {X 92.722,Y 26.2275,Z 98,A 10.4739,B 24.9232,C -2.0236,E1 25.1542,E2 74.8035} C_DIS
LIN {X 93.6503,Y 22.6914,Z 98,A 8.2896,B 24.9237,C -2.0166,E1 25.1557,E2 76.9919} C_DIS
LIN {X 94.4604,Y 19.0422,Z 98,A 6.098,B 24.9242,C -2.0109,E1 25.1569,E2 79.1842} C_DIS
LIN {X 94.9348,Y 16.5208,Z 98,A 4.1792,B 24.9257,C -1.991,E1 25.1579,E2 81.1386} C_DIS
LIN {X 95.4304,Y 13.3541,Z 98,A 2.8119,B 24.9246,C -2.0056,E1 25.1584,E2 82.4633} C_DIS
LIN {X 95.8087,Y 10.2958,Z 98,A 0.9273,B 24.9252,C -1.9978,E1 25.159,E2 84.3552} C_DIS
LIN {X 96.1117,Y 6.9263,Z 98,A -1.3598,B 24.9264,C -1.9808,E1 25.1595,E2 86.6689} C_DIS
LIN {X 96.3153,Y 2.9345,Z 98,A -3.7426,B 24.927,C -1.973,E1 25.1598,E2 89.056} C_DIS
LIN {X 96.3536,Y -1.2322,Z 98,A -5.9697,B 24.9269,C -1.9746,E1 25.1598,E2 91.2661} C_DIS
LIN {X 96.2524,Y -4.5731,Z 98,A -8.0716,B 24.9277,C -1.9638,E1 25.1595,E2 93.381} C_DIS
LIN {X 95.9271,Y -9.1273,Z 98,A -10.5098,B 24.9276,C -1.9657,E1 25.159,E2 95.8002} C_DIS
LIN {X 95.5813,Y -12.2268,Z 98,A -12.3897,B 24.9281,C -1.9587,E1 25.1583,E2 97.6854} C_DIS
LIN {X 95.1011,Y -15.5297,Z 98,A -14.4349,B 24.9287,C -1.95,E1 25.1575,E2 99.7392} C_DIS
LIN {X 94.2753,Y -19.9434,Z 98,A -17.2352,B 24.9297,C -1.9364,E1 25.1559,E2 102.5552} C_DIS
LIN {X 93.3497,Y -23.8975,Z 98,A -19.4078,B 24.9296,C -1.9381,E1 25.1545,E2 104.7112} C_DIS
LIN {X 92.6197,Y -26.5885,Z 98,A -21.9284,B 24.9323,C -1.8998,E1 25.1525,E2 107.3077} C_DIS
LIN {X 91.1962,Y -31.1228,Z 98,A -23.9659,B 24.9308,C -1.9211,E1 25.1508,E2 109.2834} C_DIS
LIN {X 90.0075,Y -34.4093,Z 98,A -25.7668,B 24.9305,C -1.9254,E1 25.149,E2 111.0643} C_DIS
LIN {X 88.4927,Y -38.1372,Z 98,A -28.3543,B 24.9316,C -1.9105,E1 25.1462,E2 113.6726} C_DIS
LIN {X 87.0652,Y -41.2933,Z 98,A -30.3367,B 24.9318,C -1.9073,E1 25.1439,E2 115.6519} C_DIS
LIN {X 85.1203,Y -45.1648,Z 98,A -33.0078,B 24.9326,C -1.896,E1 25.1405,E2 118.3354} C_DIS
LIN {X 83.3102,Y -48.424,Z 98,A -35.1576,B 24.9329,C -1.8921,E1 25.1375,E2 120.4833} C_DIS
LIN {X 81.577,Y -51.2886,Z 98,A -37.973,B 24.9355,C -1.8551,E1 25.1333,E2 123.3718} C_DIS
LIN {X 78.9277,Y -55.2791,Z 98,A -39.5919,B 24.9328,C -1.8939,E1 25.1309,E2 124.891} C_DIS
LIN {X 75.8746,Y -59.4011,Z 98,A -42.951,B 24.9342,C -1.8738,E1 25.1252,E2 128.2816} C_DIS
LIN {X 71.864,Y -64.1937,Z 98,A -46.7484,B 24.9351,C -1.861,E1 25.1183,E2 132.0919} C_DIS
LIN {X 68.7695,Y -67.4989,Z 98,A -49.3487,B 24.9353,C -1.8578,E1 25.1133,E2 134.6885} C_DIS
LIN {X 66.9766,Y -69.2777,Z 98,A -51.5228,B 24.9373,C -1.8289,E1 25.1088,E2 136.9218} C_DIS
LIN {X 63.9199,Y -72.109,Z 98,A -54.1833,B 24.9382,C -1.8163,E1 25.1032,E2 139.6015} C_DIS
LIN {X 60.2056,Y -75.2388,Z 98,A -56.255,B 24.9365,C -1.8404,E1 25.0989,E2 141.6084} C_DIS
LIN {X 55.0947,Y -79.0559,Z 98,A -59.5768,B 24.9358,C -1.8502,E1 25.0915,E2 144.8951} C_DIS
LIN {X 52.595,Y -80.7422,Z 98,A -61.8249,B 24.9373,C -1.8296,E1 25.0862,E2 147.1846} C_DIS
LIN {X 49.3771,Y -82.7485,Z 98,A -64.4195,B 24.9384,C -1.8127,E1 25.0799,E2 149.8109} C_DIS
LIN {X 46.5904,Y -84.3492,Z 98,A -66.0276,B 24.9379,C -1.8206,E1 25.076,E2 151.3957} C_DIS
LIN {X 43.3958,Y -86.0367,Z 98,A -68.0617,B 24.9379,C -1.8212,E1 25.071,E2 153.4227} C_DIS
LIN {X 39.4896,Y -87.8967,Z 98,A -70.7418,B 24.9384,C -1.8132,E1 25.0642,E2 156.1148} C_DIS
LIN {X 34.7618,Y -89.8723,Z 98,A -73.8213,B 24.9388,C -1.8077,E1 25.0562,E2 159.2005} C_DIS
LIN {X 31.2489,Y -91.1537,Z 98,A -76.1837,B 24.9393,C -1.7997,E1 25.0499,E2 161.5769} C_DIS
LIN {X 26.6137,Y -92.6126,Z 98,A -78.7551,B 24.9387,C -1.808,E1 25.0431,E2 164.1242} C_DIS
LIN {X 23.4513,Y -93.4644,Z 98,A -80.8029,B 24.9391,C -1.8023,E1 25.0375,E2 166.1823} C_DIS
LIN {X 19.6304,Y -94.3396,Z 98,A -82.6986,B 24.9382,C -1.816,E1 25.0325,E2 168.0429} C_DIS
LIN {X 16.3184,Y -94.9692,Z 98,A -85.0515,B 24.9392,C -1.8017,E1 25.0259,E2 170.4272} C_DIS
LIN {X 12.9147,Y -95.4921,Z 98,A -87.1647,B 24.9394,C -1.798,E1 25.0201,E2 172.5474} C_DIS
LIN {X 8.7778,Y -95.9594,Z 98,A -89.8281,B 24.94,C -1.7899,E1 25.0126,E2 175.2282} C_DIS
LIN {X 4.0536,Y -96.2747,Z 98,A -92.2919,B 24.9392,C -1.8013,E1 25.0058,E2 177.6641} C_DIS
LIN {X 0.6886,Y -96.3576,Z 98,A -93.4685,B 24.9372,C -1.8304,E1 25.0028,E2 178.7715} C_DIS
Enddeposition()
LIN {X 0.6886,Y -96.3576,Z 98,A -93.4685,B 24.9372,C -1.8304,E1 25.0028,E2 178.7715} C_DIS
Startdeposition()
$VEL.CP = VEL_PRINT
LIN {X 1.9855,Y -95.4441,Z 98,A -92.6473,B 24.936,C -1.8476,E1 25.0051,E2 177.9096} C_DIS
LIN {X 5.4788,Y -95.3074,Z 98,A -90.5183,B 24.9359,C -1.8495,E1 25.0111,E2 175.7768} C_DIS
LIN {X 9.5919,Y -94.9821,Z 98,A -88.1501,B 24.9361,C -1.8469,E1 25.0177,E2 173.4162} C_DIS
LIN {X 12.5815,Y -94.6323,Z 98,A -86.2285,B 24.9357,C -1.8522,E1 25.023,E2 171.4835} C_DIS
LIN {X 15.991,Y -94.116,Z 98,A -84.3639,B 24.9361,C -1.8463,E1 25.0281,E2 169.6348} C_DIS
LIN {X 19.0249,Y -93.5498,Z 98,A -82.3479,B 24.9356,C -1.8538,E1 25.0337,E2 167.6033} C_DIS
LIN {X 22.8708,Y -92.6848,Z 98,A -80.1424,B 24.9358,C -1.8502,E1 25.0396,E2 165.4095} C_DIS
LIN {X 25.7421,Y -91.9288,Z 98,A -78.3276,B 24.9356,C -1.8533,E1 25.0445,E2 163.5902} C_DIS
LIN {X 28.5928,Y -91.0826,Z 98,A -75.7125,B 24.9333,C -1.8862,E1 25.0517,E2 160.902} C_DIS
LIN {X 32.7527,Y -89.6702,Z 98,A -72.9633,B 24.9328,C -1.8939,E1 25.0589,E2 158.1403} C_DIS
LIN {X 37.2771,Y -87.886,Z 98,A -70.4283,B 24.9335,C -1.8837,E1 25.0654,E2 155.6353} C_DIS
LIN {X 40.4647,Y -86.4645,Z 98,A -68.9149,B 24.9348,C -1.8652,E1 25.0691,E2 154.1695} C_DIS
LIN {X 43.4719,Y -84.9922,Z 98,A -66.8964,B 24.9345,C -1.8689,E1 25.0742,E2 152.1479} C_DIS
LIN {X 46.4193,Y -83.4191,Z 98,A -64.8678,B 24.9342,C -1.8732,E1 25.0791,E2 150.1148} C_DIS
LIN {X 48.735,Y -82.0878,Z 98,A -63.2079,B 24.9339,C -1.8783,E1 25.0832,E2 148.4479} C_DIS
LIN {X 51.8129,Y -80.1809,Z 98,A -61.1647,B 24.9339,C -1.8776,E1 25.088,E2 146.4131} C_DIS
LIN {X 54.6559,Y -78.2703,Z 98,A -58.9592,B 24.9332,C -1.8873,E1 25.0931,E2 144.1919} C_DIS
LIN {X 58.9764,Y -75.0689,Z 98,A -55.364,B 24.9317,C -1.9082,E1 25.1011,E2 140.5606} C_DIS
LIN {X 61.5041,Y -73.0106,Z 98,A -53.7071,B 24.9322,C -1.9012,E1 25.1046,E2 138.9266} C_DIS
LIN {X 64.9843,Y -69.9314,Z 98,A -50.7997,B 24.9315,C -1.9122,E1 25.1107,E2 136.0049} C_DIS
LIN {X 67.5564,Y -67.4528,Z 98,A -48.5015,B 24.9307,C -1.9233,E1 25.1153,E2 133.6902} C_DIS
LIN {X 69.8037,Y -65.1212,Z 98,A -46.9112,B 24.9313,C -1.9146,E1 25.1182,E2 132.1274} C_DIS
LIN {X 72.642,Y -61.9404,Z 98,A -44.2544,B 24.9305,C -1.925,E1 25.1231,E2 129.4581} C_DIS
LIN {X 75.2609,Y -58.7334,Z 98,A -41.2642,B 24.9286,C -1.9511,E1 25.1284,E2 126.4203} C_DIS
LIN {X 77.8577,Y -55.2424,Z 98,A -39.2067,B 24.9297,C -1.9368,E1 25.1316,E2 124.4064} C_DIS
LIN {X 80.5403,Y -51.253,Z 98,A -36.8839,B 24.9307,C -1.9233,E1 25.1352,E2 122.1272} C_DIS
LIN {X 82.5031,Y -48.0313,Z 98,A -34.2833,B 24.9292,C -1.9427,E1 25.1389,E2 119.494} C_DIS
LIN {X 84.0029,Y -45.3544,Z 98,A -32.4143,B 24.9288,C -1.9492,E1 25.1414,E2 117.6196} C_DIS
LIN {X 85.8476,Y -41.7597,Z 98,A -30.069,B 24.9285,C -1.9533,E1 25.1444,E2 115.277} C_DIS
LIN {X 87.2534,Y -38.7376,Z 98,A -27.9722,B 24.9277,C -1.9631,E1 25.1468,E2 113.1686} C_DIS
LIN {X 89.1894,Y -34.0409,Z 98,A -25.3724,B 24.9283,C -1.955,E1 25.1495,E2 110.602} C_DIS
LIN {X 90.0517,Y -31.6888,Z 98,A -22.6008,B 24.9243,C -2.0091,E1 25.1522,E2 107.7183} C_DIS
LIN {X 91.6378,Y -26.761,Z 98,A -20.484,B 24.9265,C -1.9801,E1 25.1538,E2 105.682} C_DIS
LIN {X 92.4914,Y -23.6395,Z 98,A -18.4929,B 24.9259,C -1.9882,E1 25.1552,E2 103.6834} C_DIS
LIN {X 93.3138,Y -20.1507,Z 98,A -16.3912,B 24.9255,C -1.9931,E1 25.1565,E2 101.5823} C_DIS
LIN {X 93.8514,Y -17.4849,Z 98,A -14.6717,B 24.9249,C -2.0017,E1 25.1574,E2 99.8526} C_DIS
LIN {X 94.4294,Y -14.0311,Z 98,A -12.5802,B 24.9244,C -2.0081,E1 25.1583,E2 97.7584} C_DIS
LIN {X 94.9206,Y -10.179,Z 98,A -10.3392,B 24.9241,C -2.0121,E1 25.159,E2 95.5211} C_DIS
LIN {X 95.2271,Y -6.7347,Z 98,A -8.4494,B 24.9241,C -2.0116,E1 25.1595,E2 93.6436} C_DIS
LIN {X 95.3764,Y -4.1009,Z 98,A -6.767,B 24.9234,C -2.0206,E1 25.1597,E2 91.9502} C_DIS
LIN {X 95.4616,Y -0.7708,Z 98,A -4.7085,B 24.9228,C -2.0293,E1 25.1597,E2 89.8832} C_DIS
LIN {X 95.4288,Y 2.6293,Z 98,A -3.001,B 24.9233,C -2.023,E1 25.1597,E2 88.2009} C_DIS
LIN {X 95.3037,Y 5.5457,Z 98,A -0.9184,B 24.9219,C -2.0414,E1 25.1594,E2 86.0873} C_DIS
LIN {X 95.0027,Y 9.395,Z 98,A 1.4144,B 24.9212,C -2.0493,E1 25.1588,E2 83.7495} C_DIS
LIN {X 94.5918,Y 12.8903,Z 98,A 3.3279,B 24.9213,C -2.0483,E1 25.1582,E2 81.8497} C_DIS
LIN {X 94.1266,Y 15.9279,Z 98,A 5.2612,B 24.9206,C -2.0576,E1 25.1573,E2 79.9059} C_DIS
LIN {X 93.5002,Y 19.2661,Z 98,A 7.1683,B 24.9206,C -2.0589,E1 25.1563,E2 78.0069} C_DIS
LIN {X 92.7743,Y 22.5037,Z 98,A 9.2164,B 24.9199,C -2.0672,E1 25.155,E2 75.951} C_DIS
LIN {X 91.8826,Y 25.9049,Z 98,A 11.2883,B 24.9195,C -2.0721,E1 25.1535,E2 73.8794} C_DIS
LIN {X 90.8916,Y 29.1931,Z 98,A 13.2177,B 24.9194,C -2.0733,E1 25.1519,E2 71.9582} C_DIS
LIN {X 89.3301,Y 33.6694,Z 98,A 15.8322,B 24.9194,C -2.0728,E1 25.1495,E2 69.3595} C_DIS
LIN {X 88.5406,Y 35.6952,Z 98,A 17.5081,B 24.918,C -2.0908,E1 25.1477,E2 67.6504} C_DIS
LIN {X 87.1802,Y 38.9001,Z 98,A 19.8082,B 24.9169,C -2.1049,E1 25.1451,E2 65.3296} C_DIS
LIN {X 85.4559,Y 42.5535,Z 98,A 21.8884,B 24.9174,C -2.0985,E1 25.1426,E2 63.2757} C_DIS
LIN {X 84.0727,Y 45.2258,Z 98,A 23.853,B 24.9165,C -2.1095,E1 25.14,E2 61.2954} C_DIS
LIN {X 82.222,Y 48.5079,Z 98,A 26.0355,B 24.9163,C -2.1126,E1 25.137,E2 59.117} C_DIS
LIN {X 80.3293,Y 51.5818,Z 98,A 28.1193,B 24.9161,C -2.1151,E1 25.1339,E2 57.0378} C_DIS
LIN {X 78.0544,Y 54.9665,Z 98,A 30.5053,B 24.9158,C -2.1189,E1 25.1301,E2 54.6545} C_DIS
LIN {X 76.299,Y 57.3754,Z 98,A 32.3547,B 24.9153,C -2.1257,E1 25.127,E2 52.7981} C_DIS
LIN {X 73.8757,Y 60.4654,Z 98,A 34.5956,B 24.9152,C -2.1269,E1 25.1232,E2 50.5647} C_DIS
LIN {X 72.2326,Y 62.4194,Z 98,A 36.3512,B 24.9142,C -2.1388,E1 25.1199,E2 48.7889} C_DIS
LIN {X 69.8515,Y 65.0726,Z 98,A 38.657,B 24.9133,C -2.1499,E1 25.1156,E2 46.4671} C_DIS
LIN {X 67.1481,Y 67.8573,Z 98,A 40.7278,B 24.9137,C -2.1452,E1 25.1115,E2 44.4163} C_DIS
LIN {X 61.7252,Y 72.8254,Z 98,A 45.1669,B 24.9129,C -2.1548,E1 25.1023,E2 39.972} C_DIS
LIN {X 59.0694,Y 74.9954,Z 98,A 47.1802,B 24.9127,C -2.157,E1 25.0979,E2 37.9613} C_DIS
LIN {X 55.5507,Y 77.6377,Z 98,A 49.4078,B 24.9136,C -2.1464,E1 25.093,E2 35.7667} C_DIS
LIN {X 53.5828,Y 79.0086,Z 98,A 51.2147,B 24.9123,C -2.1622,E1 25.0888,E2 33.9284} C_DIS
LIN {X 50.0889,Y 81.2706,Z 98,A 53.8207,B 24.9117,C -2.1701,E1 25.0826,E2 31.3124} C_DIS
LIN {X 47.1372,Y 83.0169,Z 98,A 55.8266,B 24.9116,C -2.1711,E1 25.0777,E2 29.3101} C_DIS
LIN {X 43.773,Y 84.8383,Z 98,A 57.8068,B 24.9123,C -2.1626,E1 25.0729,E2 27.3554} C_DIS
LIN {X 41.5568,Y 85.9451,Z 98,A 59.5237,B 24.9114,C -2.1729,E1 25.0686,E2 25.619} C_DIS
LIN {X 38.3532,Y 87.4217,Z 98,A 61.7049,B 24.9111,C -2.1776,E1 25.063,E2 23.4319} C_DIS
LIN {X 34.7792,Y 88.9039,Z 98,A 63.9342,B 24.9111,C -2.1766,E1 25.0573,E2 21.2101} C_DIS
LIN {X 31.9165,Y 89.9718,Z 98,A 65.8703,B 24.9107,C -2.182,E1 25.0521,E2 19.2652} C_DIS
LIN {X 27.7098,Y 91.3563,Z 98,A 69.1652,B 24.9086,C -2.207,E1 25.0432,E2 15.917} C_DIS
LIN {X 23.7232,Y 92.4699,Z 98,A 70.8727,B 24.9108,C -2.1806,E1 25.0388,E2 14.2747} C_DIS
LIN {X 20.4569,Y 93.247,Z 98,A 72.9689,B 24.9105,C -2.1846,E1 25.0331,E2 12.172} C_DIS
LIN {X 17.2227,Y 93.8987,Z 98,A 74.9521,B 24.9105,C -2.1855,E1 25.0276,E2 10.1889} C_DIS
LIN {X 13.599,Y 94.4911,Z 98,A 77.1169,B 24.9105,C -2.1848,E1 25.0217,E2 8.0279} C_DIS
LIN {X 10.0784,Y 94.9311,Z 98,A 79.0479,B 24.911,C -2.1782,E1 25.0164,E2 6.114} C_DIS
LIN {X 7.4911,Y 95.1702,Z 98,A 80.7166,B 24.9107,C -2.1821,E1 25.0117,E2 4.4368} C_DIS
LIN {X 4.5521,Y 95.357,Z 98,A 82.6812,B 24.9101,C -2.189,E1 25.0062,E2 2.4566} C_DIS
LIN {X 1.2924,Y 95.4569,Z 98,A 84.5399,B 24.9104,C -2.1853,E1 25.001,E2 0.607} C_DIS
LIN {X -1.788,Y 95.4478,Z 98,A 86.1801,B 24.9111,C -2.1776,E1 24.9965,E2 -1.015} C_DIS
LIN {X -4.5845,Y 95.3556,Z 98,A 88.0636,B 24.9105,C -2.1841,E1 24.9912,E2 -2.9143} C_DIS
LIN {X -7.9581,Y 95.1329,Z 98,A 89.9784,B 24.9109,C -2.1793,E1 24.9859,E2 -4.8185} C_DIS
LIN {X -10.9744,Y 94.8317,Z 98,A 92.1406,B 24.91,C -2.1902,E1 24.9798,E2 -7.0078} C_DIS
LIN {X -14.8962,Y 94.2957,Z 98,A 94.334,B 24.9107,C -2.1823,E1 24.9738,E2 -9.1844} C_DIS
LIN {X -18.4604,Y 93.6636,Z 98,A 96.3854,B 24.9111,C -2.1765,E1 24.9682,E2 -11.224} C_DIS
LIN {X -21.8542,Y 92.9301,Z 98,A 98.4381,B 24.9114,C -2.1736,E1 24.9626,E2 -13.2724} C_DIS
LIN {X -26.523,Y 91.7064,Z 98,A 101.7874,B 24.9104,C -2.1859,E1 24.9535,E2 -16.6564} C_DIS
LIN {X -30.5669,Y 90.4386,Z 98,A 104.6507,B 24.9097,C -2.1938,E1 24.9458,E2 -19.5436} C_DIS
LIN {X -34.3102,Y 89.0874,Z 98,A 106.445,B 24.9116,C -2.1705,E1 24.9413,E2 -21.2862} C_DIS
LIN {X -37.25,Y 87.8974,Z 98,A 108.3561,B 24.9118,C -2.1681,E1 24.9364,E2 -23.1959} C_DIS
LIN {X -40.6268,Y 86.3891,Z 98,A 111.0573,B 24.9108,C -2.1808,E1 24.9294,E2 -25.9342} C_DIS
LIN {X -43.713,Y 84.8689,Z 98,A 112.7107,B 24.9122,C -2.1637,E1 24.9254,E2 -27.5512} C_DIS
LIN {X -47.1134,Y 83.0306,Z 98,A 114.9727,B 24.9127,C -2.1577,E1 24.9199,E2 -29.8056} C_DIS
LIN {X -50.0855,Y 81.2727,Z 98,A 117.1568,B 24.9127,C -2.1577,E1 24.9147,E2 -31.9962} C_DIS
LIN {X -52.7968,Y 79.5365,Z 98,A 119.061,B 24.9131,C -2.153,E1 24.9102,E2 -33.8956} C_DIS
LIN {X -55.921,Y 77.3735,Z 98,A 121.2927,B 24.9136,C -2.1468,E1 24.9052,E2 -36.1201} C_DIS
LIN {X -58.4482,Y 75.4807,Z 98,A 123.1966,B 24.9139,C -2.1431,E1 24.9009,E2 -38.0222} C_DIS
LIN {X -61.0587,Y 73.3847,Z 98,A 125.114,B 24.9145,C -2.1357,E1 24.8968,E2 -39.9292} C_DIS
LIN {X -63.5448,Y 71.2429,Z 98,A 127.1759,B 24.9145,C -2.1343,E1 24.8925,E2 -41.9958} C_DIS
LIN {X -66.145,Y 68.8356,Z 98,A 129.2968,B 24.915,C -2.1291,E1 24.8882,E2 -44.1131} C_DIS
LIN {X -68.647,Y 66.3406,Z 98,A 131.4221,B 24.9154,C -2.1241,E1 24.884,E2 -46.2355} C_DIS
LIN {X -71.0396,Y 63.7719,Z 98,A 133.5449,B 24.9158,C -2.1193,E1 24.88,E2 -48.3564} C_DIS
LIN {X -73.6167,Y 60.7795,Z 98,A 135.8358,B 24.9165,C -2.1106,E1 24.8759,E2 -50.637} C_DIS
LIN {X -75.3335,Y 58.6393,Z 98,A 137.6707,B 24.9163,C -2.1124,E1 24.8727,E2 -52.4847} C_DIS
LIN {X -77.2912,Y 56.0334,Z 98,A 139.4362,B 24.9172,C -2.1009,E1 24.8698,E2 -54.2314} C_DIS
LIN {X -78.9688,Y 53.6416,Z 98,A 141.3385,B 24.9172,C -2.1009,E1 24.8668,E2 -56.143} C_DIS
LIN {X -80.4569,Y 51.383,Z 98,A 142.8477,B 24.9179,C -2.0927,E1 24.8645,E2 -57.6403} C_DIS
LIN {X -81.8334,Y 49.1631,Z 98,A 144.4516,B 24.9181,C -2.0894,E1 24.8622,E2 -59.2445} C_DIS
LIN {X -83.3175,Y 46.6013,Z 98,A 146.3872,B 24.9181,C -2.0894,E1 24.8595,E2 -61.1901} C_DIS
LIN {X -85.2388,Y 42.9893,Z 98,A 149.0323,B 24.9182,C -2.0882,E1 24.8561,E2 -63.8466} C_DIS
LIN {X -87.7037,Y 37.7063,Z 98,A 152.1912,B 24.9199,C -2.0668,E1 24.8525,E2 -66.9717} C_DIS
LIN {X -88.8376,Y 34.948,Z 98,A 154.1382,B 24.9199,C -2.0663,E1 24.8504,E2 -68.9285} C_DIS
LIN {X -90.0141,Y 31.7959,Z 98,A 156.1854,B 24.9203,C -2.061,E1 24.8485,E2 -70.9746} C_DIS
LIN {X -91.0619,Y 28.6596,Z 98,A 157.9998,B 24.9212,C -2.0494,E1 24.8469,E2 -72.7716} C_DIS
LIN {X -91.8546,Y 26.0041,Z 98,A 160.0352,B 24.9207,C -2.056,E1 24.8453,E2 -74.8347} C_DIS
LIN {X -92.637,Y 23.0667,Z 98,A 161.7428,B 24.9215,C -2.0465,E1 24.8442,E2 -76.5295} C_DIS
LIN {X -93.4075,Y 19.7179,Z 98,A 163.8641,B 24.9218,C -2.0418,E1 24.8429,E2 -78.6521} C_DIS
LIN {X -94.0486,Y 16.3893,Z 98,A 166.4262,B 24.921,C -2.0522,E1 24.8416,E2 -81.2542} C_DIS
LIN {X -94.6334,Y 12.5729,Z 98,A 167.8449,B 24.9238,C -2.0161,E1 24.8411,E2 -82.5952} C_DIS
LIN {X -95.0581,Y 8.8,Z 98,A 170.356,B 24.9238,C -2.0161,E1 24.8404,E2 -85.1214} C_DIS
LIN {X -95.3062,Y 5.5014,Z 98,A 172.4067,B 24.9241,C -2.0118,E1 24.84,E2 -87.1742} C_DIS
LIN {X -95.4306,Y 2.5683,Z 98,A 174.4977,B 24.9237,C -2.0166,E1 24.8398,E2 -89.2892} C_DIS
LIN {X -95.4608,Y -0.9068,Z 98,A 176.3574,B 24.9248,C -2.0027,E1 24.8398,E2 -91.127} C_DIS
LIN {X -95.2746,Y -6.0321,Z 98,A 179.3398,B 24.9258,C -1.9898,E1 24.8402,E2 -94.0965} C_DIS
LIN {X -95.0395,Y -9.0011,Z 98,A -178.7162,B 24.9258,C -1.9891,E1 24.8407,E2 -96.0504} C_DIS
LIN {X -94.6677,Y -12.3082,Z 98,A -176.8229,B 24.9265,C -1.9795,E1 24.8413,E2 -97.9322} C_DIS
LIN {X -93.7987,Y -17.7584,Z 98,A -172.709,B 24.9254,C -1.9949,E1 24.8433,E2 -102.1073} C_DIS
LIN {X -92.8898,Y -22.0288,Z 98,A -169.6416,B 24.9249,C -2.0015,E1 24.8454,E2 -105.2082} C_DIS
LIN {X -91.3646,Y -27.6818,Z 98,A -167.41,B 24.9288,C -1.9491,E1 24.847,E2 -107.328} C_DIS
LIN {X -90.3557,Y -30.8128,Z 98,A -165.2053,B 24.9287,C -1.9507,E1 24.849,E2 -109.5489} C_DIS
LIN {X -89.168,Y -34.0974,Z 98,A -163.0861,B 24.9291,C -1.9453,E1 24.851,E2 -111.6671} C_DIS
LIN {X -87.8958,Y -37.2538,Z 98,A -161.0306,B 24.9295,C -1.9398,E1 24.8532,E2 -113.7211} C_DIS
LIN {X -86.3024,Y -40.813,Z 98,A -158.6777,B 24.9299,C -1.9336,E1 24.856,E2 -116.0719} C_DIS
LIN {X -84.783,Y -43.8813,Z 98,A -156.3798,B 24.9297,C -1.9358,E1 24.8589,E2 -118.3876} C_DIS
LIN {X -83.0265,Y -47.1205,Z 98,A -154.3765,B 24.9307,C -1.923,E1 24.8616,E2 -120.3709} C_DIS
LIN {X -81.1031,Y -50.3569,Z 98,A -152.197,B 24.9313,C -1.9145,E1 24.8648,E2 -122.5412} C_DIS
LIN {X -79.2483,Y -53.2288,Z 98,A -150.098,B 24.9316,C -1.9108,E1 24.868,E2 -124.6418} C_DIS
LIN {X -77.1413,Y -56.2382,Z 98,A -148.2,B 24.9327,C -1.8953,E1 24.871,E2 -126.5121} C_DIS
LIN {X -75.7395,Y -58.1124,Z 98,A -146.5441,B 24.9323,C -1.9001,E1 24.8738,E2 -128.1874} C_DIS
LIN {X -73.6699,Y -60.7155,Z 98,A -144.4723,B 24.9325,C -1.8979,E1 24.8775,E2 -130.2636} C_DIS
LIN {X -71.419,Y -63.3482,Z 98,A -142.1125,B 24.9321,C -1.9025,E1 24.8819,E2 -132.645} C_DIS
LIN {X -68.1614,Y -66.8403,Z 98,A -139.5213,B 24.9332,C -1.8871,E1 24.8868,E2 -135.2108} C_DIS
LIN {X -64.5513,Y -70.3321,Z 98,A -136.6028,B 24.9339,C -1.8777,E1 24.8927,E2 -138.119} C_DIS
LIN {X -62.263,Y -72.3672,Z 98,A -134.6412,B 24.9339,C -1.8782,E1 24.8968,E2 -140.0895} C_DIS
LIN {X -59.625,Y -74.5563,Z 98,A -132.4163,B 24.9337,C -1.88,E1 24.9017,E2 -142.3272} C_DIS
LIN {X -56.6249,Y -76.8582,Z 98,A -130.3013,B 24.9344,C -1.8709,E1 24.9064,E2 -144.4279} C_DIS
LIN {X -53.5657,Y -79.0202,Z 98,A -128.1351,B 24.9348,C -1.8644,E1 24.9113,E2 -146.5861} C_DIS
LIN {X -50.9598,Y -80.7266,Z 98,A -126.1302,B 24.9348,C -1.8661,E1 24.9161,E2 -148.6014} C_DIS
LIN {X -48.0231,Y -82.5078,Z 98,A -123.9466,B 24.9346,C -1.8673,E1 24.9213,E2 -150.7944} C_DIS
LIN {X -44.4793,Y -84.4693,Z 98,A -121.6819,B 24.9353,C -1.8584,E1 24.9269,E2 -153.0445} C_DIS
LIN {X -41.3074,Y -86.065,Z 98,A -119.5893,B 24.9355,C -1.8545,E1 24.9321,E2 -155.1332} C_DIS
LIN {X -37.9458,Y -87.5993,Z 98,A -117.5255,B 24.9361,C -1.8467,E1 24.9373,E2 -157.1836} C_DIS
LIN {X -35.5859,Y -88.5851,Z 98,A -115.7384,B 24.9356,C -1.8538,E1 24.942,E2 -158.9916} C_DIS
LIN {X -32.431,Y -89.7875,Z 98,A -113.6909,B 24.9356,C -1.8528,E1 24.9474,E2 -161.0408} C_DIS
LIN {X -26.7732,Y -91.6342,Z 98,A -110.2394,B 24.9361,C -1.8459,E1 24.9565,E2 -164.482} C_DIS
LIN {X -23.5151,Y -92.5234,Z 98,A -108.1302,B 24.9361,C -1.8475,E1 24.9622,E2 -166.5983} C_DIS
LIN {X -20.5294,Y -93.2312,Z 98,A -106.3067,B 24.9361,C -1.846,E1 24.9672,E2 -168.4205} C_DIS
LIN {X -17.2254,Y -93.8982,Z 98,A -104.2179,B 24.9361,C -1.8475,E1 24.973,E2 -170.5152} C_DIS
LIN {X -13.9542,Y -94.4407,Z 98,A -102.2962,B 24.9362,C -1.8446,E1 24.9782,E2 -172.4315} C_DIS
LIN {X -10.8921,Y -94.8413,Z 98,A -100.5368,B 24.9365,C -1.8409,E1 24.9831,E2 -174.1837} C_DIS
LIN {X -7.6886,Y -95.1544,Z 98,A -98.4657,B 24.9361,C -1.8458,E1 24.9889,E2 -176.2672} C_DIS
LIN {X -4.1127,Y -95.3759,Z 98,A -96.3426,B 24.9361,C -1.8449,E1 24.9948,E2 -178.3889} C_DIS
LIN {X -0.5162,Y -95.4631,Z 98,A -94.4195,B 24.9368,C -1.8369,E1 25.0001,E2 -180.293} C_DIS
LIN {X -0.5162,Y -95.4631,Z 98,A -94.4195,B 24.9368,C -1.8369,E1 25.0001,E2 -180.293} C_DIS
Enddeposition()
LIN {X 0.6693,Y -94.5646,Z 98,A -93.8393,B 24.936,C -1.848,E1 25.0018,E2 -180.8996} C_DIS
Startdeposition()
$VEL.CP = VEL_PRINT
LIN {X -1.5836,Y -94.5559,Z 98,A -95.7401,B 24.9373,C -1.8289,E1 24.9964,E2 -178.9535} C_DIS
LIN {X -4.6527,Y -94.4562,Z 98,A -97.692,B 24.9375,C -1.8255,E1 24.9909,E2 -176.993} C_DIS
LIN {X -7.3776,Y -94.281,Z 98,A -99.2546,B 24.9373,C -1.8287,E1 24.9866,E2 -175.4374} C_DIS
LIN {X -10.4241,Y -93.9946,Z 98,A -101.1885,B 24.9375,C -1.8261,E1 24.9812,E2 -173.4962} C_DIS
LIN {X -13.4778,Y -93.6039,Z 98,A -102.9472,B 24.9372,C -1.8302,E1 24.9763,E2 -171.7458} C_DIS
LIN {X -16.4453,Y -93.1286,Z 98,A -104.7587,B 24.9372,C -1.831,E1 24.9714,E2 -169.9347} C_DIS
LIN {X -19.182,Y -92.6033,Z 98,A -106.4565,B 24.9372,C -1.8314,E1 24.9667,E2 -168.2359} C_DIS
LIN {X -21.849,Y -92.0123,Z 98,A -108.2229,B 24.9373,C -1.8284,E1 24.9619,E2 -166.46} C_DIS
LIN {X -24.5108,Y -91.3375,Z 98,A -109.8254,B 24.9371,C -1.8315,E1 24.9576,E2 -164.8625} C_DIS
LIN {X -27.4961,Y -90.4851,Z 98,A -111.7603,B 24.9371,C -1.8309,E1 24.9524,E2 -162.9231} C_DIS
LIN {X -30.4674,Y -89.5272,Z 98,A -113.712,B 24.9371,C -1.8304,E1 24.9472,E2 -160.9664} C_DIS
LIN {X -33.6532,Y -88.3787,Z 98,A -115.6138,B 24.9367,C -1.8373,E1 24.9422,E2 -159.0772} C_DIS
LIN {X -36.189,Y -87.3727,Z 98,A -117.2096,B 24.9365,C -1.8408,E1 24.9381,E2 -157.4862} C_DIS
LIN {X -38.7113,Y -86.2831,Z 98,A -118.8777,B 24.9364,C -1.8425,E1 24.9338,E2 -155.8183} C_DIS
LIN {X -41.1102,Y -85.1662,Z 98,A -120.5477,B 24.9364,C -1.8422,E1 24.9296,E2 -154.1431} C_DIS
LIN {X -43.9226,Y -83.7504,Z 98,A -122.4905,B 24.9364,C -1.8434,E1 24.9248,E2 -152.198} C_DIS
LIN {X -46.6245,Y -82.2787,Z 98,A -124.2663,B 24.9359,C -1.8489,E1 24.9205,E2 -150.43} C_DIS
LIN {X -48.6236,Y -81.1133,Z 98,A -125.8445,B 24.9362,C -1.8451,E1 24.9166,E2 -148.838} C_DIS
LIN {X -51.2192,Y -79.4979,Z 98,A -127.5948,B 24.9358,C -1.8513,E1 24.9125,E2 -147.0969} C_DIS
LIN {X -53.5557,Y -77.9445,Z 98,A -129.3828,B 24.9358,C -1.8511,E1 24.9084,E2 -145.3026} C_DIS
LIN {X -56.0518,Y -76.1679,Z 98,A -131.3136,B 24.9358,C -1.8518,E1 24.904,E2 -143.3668} C_DIS
LIN {X -58.8115,Y -74.0578,Z 98,A -133.4251,B 24.9355,C -1.8554,E1 24.8994,E2 -141.256} C_DIS
LIN {X -61.3326,Y -71.9834,Z 98,A -135.3095,B 24.935,C -1.8622,E1 24.8953,E2 -139.3805} C_DIS
LIN {X -63.9346,Y -69.6826,Z 98,A -137.4369,B 24.9348,C -1.8656,E1 24.8909,E2 -137.2527} C_DIS
LIN {X -66.4667,Y -67.2717,Z 98,A -139.5512,B 24.9344,C -1.8701,E1 24.8867,E2 -135.1404} C_DIS
LIN {X -68.8877,Y -64.7904,Z 98,A -141.4805,B 24.9337,C -1.8802,E1 24.883,E2 -133.2267} C_DIS
LIN {X -70.4657,Y -63.0705,Z 98,A -143.0847,B 24.9339,C -1.8772,E1 24.8799,E2 -131.6083} C_DIS
LIN {X -72.7347,Y -60.4398,Z 98,A -145.1988,B 24.9336,C -1.8818,E1 24.8761,E2 -129.4954} C_DIS
LIN {X -74.9056,Y -57.7274,Z 98,A -147.316,B 24.9333,C -1.8864,E1 24.8725,E2 -127.3792} C_DIS
LIN {X -76.6373,Y -55.4107,Z 98,A -149.1415,B 24.9332,C -1.8884,E1 24.8694,E2 -125.5496} C_DIS
LIN {X -78.4622,Y -52.7927,Z 98,A -151.1268,B 24.9329,C -1.8916,E1 24.8663,E2 -123.5622} C_DIS
LIN {X -80.2974,Y -49.9566,Z 98,A -153.0333,B 24.9322,C -1.9014,E1 24.8635,E2 -121.6693} C_DIS
LIN {X -81.9139,Y -47.2592,Z 98,A -154.8871,B 24.9317,C -1.9081,E1 24.8609,E2 -119.8219} C_DIS
LIN {X -83.0595,Y -45.2155,Z 98,A -156.4037,B 24.9317,C -1.9088,E1 24.8588,E2 -118.2991} C_DIS
LIN {X -84.4729,Y -42.5201,Z 98,A -158.3397,B 24.9315,C -1.911,E1 24.8563,E2 -116.3579} C_DIS
LIN {X -85.805,Y -39.7597,Z 98,A -160.2341,B 24.9312,C -1.915,E1 24.8541,E2 -114.4629} C_DIS
LIN {X -87.0862,Y -36.8691,Z 98,A -161.9663,B 24.9304,C -1.9263,E1 24.8522,E2 -112.7479} C_DIS
LIN {X -87.9631,Y -34.725,Z 98,A -163.3791,B 24.9302,C -1.9301,E1 24.8507,E2 -111.3362} C_DIS
LIN {X -88.9001,Y -32.2507,Z 98,A -165.0548,B 24.93,C -1.9325,E1 24.8491,E2 -109.6568} C_DIS
LIN {X -89.8002,Y -29.6573,Z 98,A -166.8369,B 24.9299,C -1.9337,E1 24.8475,E2 -107.8674} C_DIS
LIN {X -90.7298,Y -26.6733,Z 98,A -168.6401,B 24.9293,C -1.9422,E1 24.846,E2 -106.0742} C_DIS
LIN {X -91.4544,Y -24.0771,Z 98,A -170.3807,B 24.9292,C -1.9438,E1 24.8447,E2 -104.3274} C_DIS
LIN {X -92.1776,Y -21.1332,Z 98,A -172.2925,B 24.9289,C -1.9472,E1 24.8435,E2 -102.4123} C_DIS
LIN {X -92.8848,Y -17.769,Z 98,A -174.2304,B 24.9281,C -1.9581,E1 24.8424,E2 -100.4891} C_DIS
LIN {X -93.3531,Y -15.1236,Z 98,A -175.9813,B 24.9281,C -1.9594,E1 24.8416,E2 -98.7308} C_DIS
LIN {X -93.8054,Y -11.9951,Z 98,A -177.7982,B 24.9273,C -1.9685,E1 24.8409,E2 -96.9248} C_DIS
LIN {X -94.1539,Y -8.8527,Z 98,A -179.7527,B 24.927,C -1.9733,E1 24.8404,E2 -94.9702} C_DIS
LIN {X -94.3927,Y -5.8011,Z 98,A 178.1118,B 24.9272,C -1.9705,E1 24.84,E2 -92.8151} C_DIS
LIN {X -94.5446,Y -2.1995,Z 98,A 176.3396,B 24.9257,C -1.9903,E1 24.8398,E2 -91.0794} C_DIS
LIN {X -94.5657,Y 0.8352,Z 98,A 174.3786,B 24.9256,C -1.9924,E1 24.8398,E2 -89.1116} C_DIS
LIN {X -94.4889,Y 3.8959,Z 98,A 172.46,B 24.9253,C -1.9964,E1 24.84,E2 -87.191} C_DIS
LIN {X -94.315,Y 6.9512,Z 98,A 170.6851,B 24.9246,C -2.0048,E1 24.8403,E2 -85.4254} C_DIS
LIN {X -94.0733,Y 9.6718,Z 98,A 168.8959,B 24.9246,C -2.006,E1 24.8408,E2 -83.6283} C_DIS
LIN {X -93.7041,Y 12.7723,Z 98,A 166.9504,B 24.9242,C -2.0104,E1 24.8415,E2 -81.6816} C_DIS
LIN {X -93.2426,Y 15.7846,Z 98,A 165.1894,B 24.9236,C -2.0189,E1 24.8422,E2 -79.9306} C_DIS
LIN {X -92.7512,Y 18.4619,Z 98,A 163.5972,B 24.923,C -2.0259,E1 24.8431,E2 -78.3458} C_DIS
LIN {X -92.1795,Y 21.125,Z 98,A 161.8395,B 24.9229,C -2.0279,E1 24.8441,E2 -76.5823} C_DIS
LIN {X -91.4513,Y 24.0889,Z 98,A 160.0656,B 24.9223,C -2.036,E1 24.8453,E2 -74.8175} C_DIS
LIN {X -90.7103,Y 26.739,Z 98,A 158.2984,B 24.9221,C -2.0382,E1 24.8467,E2 -73.0452} C_DIS
LIN {X -89.7952,Y 29.6725,Z 98,A 156.3451,B 24.9219,C -2.0411,E1 24.8484,E2 -71.0878} C_DIS
LIN {X -88.8998,Y 32.2514,Z 98,A 154.7582,B 24.9213,C -2.0483,E1 24.8498,E2 -69.5091} C_DIS
LIN {X -87.6821,Y 35.4289,Z 98,A 152.6563,B 24.9209,C -2.0534,E1 24.852,E2 -67.4075} C_DIS
LIN {X -86.3523,Y 38.5575,Z 98,A 150.5751,B 24.9205,C -2.059,E1 24.8543,E2 -65.3281} C_DIS
LIN {X -84.9639,Y 41.5297,Z 98,A 148.5485,B 24.9201,C -2.0637,E1 24.8567,E2 -63.3017} C_DIS
LIN {X -83.7463,Y 43.9305,Z 98,A 146.9674,B 24.9196,C -2.07,E1 24.8588,E2 -61.7274} C_DIS
LIN {X -82.2823,Y 46.6182,Z 98,A 145.1937,B 24.919,C -2.0779,E1 24.8612,E2 -59.9631} C_DIS
LIN {X -81.1155,Y 48.62,Z 98,A 143.6082,B 24.9192,C -2.0763,E1 24.8634,E2 -58.3655} C_DIS
LIN {X -79.4836,Y 51.2416,Z 98,A 141.8321,B 24.9185,C -2.0845,E1 24.8661,E2 -56.6001} C_DIS
LIN {X -77.974,Y 53.5133,Z 98,A 140.0656,B 24.9185,C -2.0855,E1 24.8688,E2 -54.8272} C_DIS
LIN {X -76.3963,Y 55.7399,Z 98,A 138.4797,B 24.9179,C -2.0921,E1 24.8714,E2 -53.2493} C_DIS
LIN {X -74.3248,Y 58.4737,Z 98,A 136.3571,B 24.9176,C -2.0963,E1 24.875,E2 -51.1266} C_DIS
LIN {X -72.1078,Y 61.1866,Z 98,A 134.2327,B 24.9172,C -2.1017,E1 24.8788,E2 -49.0053} C_DIS
LIN {X -69.9254,Y 63.6701,Z 98,A 132.2036,B 24.9168,C -2.106,E1 24.8826,E2 -46.9772} C_DIS
LIN {X -67.6876,Y 66.0456,Z 98,A 130.1265,B 24.9167,C -2.1077,E1 24.8866,E2 -44.8952} C_DIS
LIN {X -65.194,Y 68.5081,Z 98,A 127.9972,B 24.9163,C -2.1125,E1 24.8909,E2 -42.7685} C_DIS
LIN {X -62.6369,Y 70.8537,Z 98,A 125.8699,B 24.916,C -2.1165,E1 24.8953,E2 -40.6424} C_DIS
LIN {X -59.9945,Y 73.1047,Z 98,A 123.7656,B 24.9156,C -2.1211,E1 24.8998,E2 -38.541} C_DIS
LIN {X -57.2712,Y 75.2571,Z 98,A 121.862,B 24.9148,C -2.132,E1 24.904,E2 -36.6562} C_DIS
LIN {X -55.3909,Y 76.6517,Z 98,A 120.2747,B 24.915,C -2.1295,E1 24.9076,E2 -35.0574} C_DIS
LIN {X -52.8813,Y 78.4022,Z 98,A 118.5213,B 24.9144,C -2.1364,E1 24.9116,E2 -33.3145} C_DIS
LIN {X -50.5964,Y 79.8977,Z 98,A 116.7503,B 24.9144,C -2.1358,E1 24.9157,E2 -31.5363} C_DIS
LIN {X -48.2677,Y 81.3238,Z 98,A 115.2608,B 24.9138,C -2.1441,E1 24.9193,E2 -30.0621} C_DIS
LIN {X -46.2617,Y 82.4814,Z 98,A 113.8455,B 24.9136,C -2.1462,E1 24.9227,E2 -28.6477} C_DIS
LIN {X -43.81,Y 83.8097,Z 98,A 111.938,B 24.9139,C -2.142,E1 24.9274,E2 -26.7248} C_DIS
LIN {X -41.0814,Y 85.18,Z 98,A 110.211,B 24.9134,C -2.1489,E1 24.9317,E2 -25.0097} C_DIS
LIN {X -38.311,Y 86.4632,Z 98,A 108.2748,B 24.9134,C -2.1489,E1 24.9367,E2 -23.0687} C_DIS
LIN {X -35.8021,Y 87.5302,Z 98,A 106.7874,B 24.9128,C -2.1566,E1 24.9405,E2 -21.5963} C_DIS
LIN {X -33.61,Y 88.3951,Z 98,A 105.2689,B 24.9128,C -2.1555,E1 24.9444,E2 -20.0721} C_DIS
LIN {X -30.7513,Y 89.4314,Z 98,A 103.5014,B 24.9125,C -2.1603,E1 24.9491,E2 -18.3123} C_DIS
LIN {X -27.8977,Y 90.3606,Z 98,A 101.5504,B 24.9127,C -2.158,E1 24.9543,E2 -16.3525} C_DIS
LIN {X -25.1506,Y 91.1647,Z 98,A 99.9649,B 24.9121,C -2.1648,E1 24.9585,E2 -14.7804} C_DIS
LIN {X -22.5809,Y 91.8337,Z 98,A 98.2353,B 24.9123,C -2.1624,E1 24.9632,E2 -13.0427} C_DIS
LIN {X -19.5766,Y 92.5223,Z 98,A 96.4627,B 24.9119,C -2.1671,E1 24.968,E2 -11.2791} C_DIS
LIN {X -16.8954,Y 93.0477,Z 98,A 94.8042,B 24.9119,C -2.1684,E1 24.9726,E2 -9.6218} C_DIS
LIN {X -14.2857,Y 93.484,Z 98,A 93.126,B 24.9119,C -2.167,E1 24.9772,E2 -7.9388} C_DIS
LIN {X -11.5588,Y 93.8617,Z 98,A 91.5295,B 24.9116,C -2.1703,E1 24.9816,E2 -6.3491} C_DIS
LIN {X -8.8451,Y 94.1546,Z 98,A 89.7818,B 24.9118,C -2.1681,E1 24.9865,E2 -4.595} C_DIS
LIN {X -5.4665,Y 94.4112,Z 98,A 87.6959,B 24.9118,C -2.1678,E1 24.9923,E2 -2.5077} C_DIS
LIN {X -2.325,Y 94.5422,Z 98,A 85.7378,B 24.912,C -2.1666,E1 24.9978,E2 -0.5463} C_DIS
LIN {X 0.7518,Y 94.5662,Z 98,A 83.9294,B 24.9118,C -2.1688,E1 25.0028,E2 1.2565} C_DIS
LIN {X 3.9027,Y 94.4886,Z 98,A 82.0449,B 24.9117,C -2.1699,E1 25.0081,E2 3.1381} C_DIS
LIN {X 6.9584,Y 94.3145,Z 98,A 80.2823,B 24.9114,C -2.1729,E1 25.013,E2 4.8927} C_DIS
LIN {X 9.6791,Y 94.0726,Z 98,A 78.6216,B 24.9114,C -2.1726,E1 25.0176,E2 6.5532} C_DIS
LIN {X 11.9977,Y 93.805,Z 98,A 77.1226,B 24.9117,C -2.1694,E1 25.0217,E2 8.0587} C_DIS
LIN {X 15.0287,Y 93.369,Z 98,A 75.3604,B 24.9115,C -2.172,E1 25.0266,E2 9.8129} C_DIS
LIN {X 17.7191,Y 92.8944,Z 98,A 73.6139,B 24.9118,C -2.1683,E1 25.0314,E2 11.5664} C_DIS
LIN {X 21.0323,Y 92.2009,Z 98,A 71.5211,B 24.912,C -2.1658,E1 25.0371,E2 13.6623} C_DIS
LIN {X 24.1501,Y 91.435,Z 98,A 69.5698,B 24.9121,C -2.1644,E1 25.0424,E2 15.614} C_DIS
LIN {X 26.7471,Y 90.7079,Z 98,A 67.9901,B 24.9121,C -2.1652,E1 25.0466,E2 17.1892} C_DIS
LIN {X 29.6751,Y 89.7943,Z 98,A 66.0116,B 24.9125,C -2.1595,E1 25.0519,E2 19.1775} C_DIS
LIN {X 32.9497,Y 88.6451,Z 98,A 64.129,B 24.9121,C -2.1653,E1 25.0568,E2 21.0425} C_DIS
LIN {X 35.1277,Y 87.8047,Z 98,A 62.7188,B 24.9121,C -2.164,E1 25.0605,E2 22.4526} C_DIS
LIN {X 37.2683,Y 86.9178,Z 98,A 61.1482,B 24.9128,C -2.1566,E1 25.0646,E2 24.0369} C_DIS
LIN {X 39.7616,Y 85.8041,Z 98,A 59.5755,B 24.9127,C -2.1576,E1 25.0685,E2 25.6033} C_DIS
LIN {X 42.5184,Y 84.4738,Z 98,A 57.6193,B 24.9132,C -2.1517,E1 25.0735,E2 27.5684} C_DIS
LIN {X 45.2442,Y 83.0439,Z 98,A 55.7405,B 24.9134,C -2.1487,E1 25.0781,E2 29.4489} C_DIS
LIN {X 48.2592,Y 81.3288,Z 98,A 53.8018,B 24.9132,C -2.1515,E1 25.0827,E2 31.3751} C_DIS
LIN {X 50.6019,Y 79.8941,Z 98,A 52.2049,B 24.9132,C -2.1514,E1 25.0865,E2 32.9673} C_DIS
LIN {X 52.8874,Y 78.398,Z 98,A 50.4589,B 24.9137,C -2.1455,E1 25.0906,E2 34.7214} C_DIS
LIN {X 55.4227,Y 76.6285,Z 98,A 48.6917,B 24.9137,C -2.1461,E1 25.0946,E2 36.481} C_DIS
LIN {X 57.7333,Y 74.9011,Z 98,A 46.8394,B 24.9142,C -2.1392,E1 25.0987,E2 38.3429} C_DIS
LIN {X 60.4418,Y 72.7331,Z 98,A 44.7492,B 24.9145,C -2.1357,E1 25.1033,E2 40.4334} C_DIS
LIN {X 63.1357,Y 70.4073,Z 98,A 42.5982,B 24.9148,C -2.1317,E1 25.1078,E2 42.5854} C_DIS
LIN {X 65.6384,Y 68.0801,Z 98,A 40.526,B 24.9151,C -2.1273,E1 25.112,E2 44.6594} C_DIS
LIN {X 68.1034,Y 65.6143,Z 98,A 38.4331,B 24.9154,C -2.1235,E1 25.1161,E2 46.7524} C_DIS
LIN {X 70.4637,Y 63.0728,Z 98,A 36.3454,B 24.9158,C -2.1193,E1 25.12,E2 48.8408} C_DIS
LIN {X 72.7298,Y 60.4456,Z 98,A 34.252,B 24.9161,C -2.1147,E1 25.1238,E2 50.9354} C_DIS
LIN {X 74.9103,Y 57.7214,Z 98,A 32.1496,B 24.9165,C -2.1101,E1 25.1275,E2 53.0389} C_DIS
LIN {X 76.9392,Y 54.9879,Z 98,A 30.227,B 24.9165,C -2.1101,E1 25.1306,E2 54.9521} C_DIS
LIN {X 78.4101,Y 52.8696,Z 98,A 28.5435,B 24.9172,C -2.1017,E1 25.1333,E2 56.6473} C_DIS
LIN {X 79.9023,Y 50.589,Z 98,A 26.842,B 24.9176,C -2.0955,E1 25.1359,E2 58.3549} C_DIS
LIN {X 81.326,Y 48.264,Z 98,A 25.3688,B 24.9175,C -2.0978,E1 25.138,E2 59.8151} C_DIS
LIN {X 82.4817,Y 46.2613,Z 98,A 23.9683,B 24.9178,C -2.0941,E1 25.1399,E2 61.2172} C_DIS
LIN {X 83.7524,Y 43.9188,Z 98,A 22.3092,B 24.9182,C -2.088,E1 25.1421,E2 62.8819} C_DIS
LIN {X 85.2278,Y 40.9819,Z 98,A 20.2647,B 24.9188,C -2.0804,E1 25.1446,E2 64.9333} C_DIS
LIN {X 86.6289,Y 37.931,Z 98,A 18.266,B 24.9192,C -2.076,E1 25.1469,E2 66.9317} C_DIS
LIN {X 87.962,Y 34.7278,Z 98,A 16.2812,B 24.9193,C -2.0743,E1 25.149,E2 68.9096} C_DIS
LIN {X 88.9265,Y 32.1782,Z 98,A 14.4159,B 24.9203,C -2.0614,E1 25.1508,E2 70.7949} C_DIS
LIN {X 90.0262,Y 28.9587,Z 98,A 12.5295,B 24.9203,C -2.0618,E1 25.1525,E2 72.6697} C_DIS
LIN {X 90.9406,Y 25.9447,Z 98,A 10.5843,B 24.9208,C -2.0546,E1 25.154,E2 74.6207} C_DIS
LIN {X 91.8375,Y 22.5653,Z 98,A 8.5016,B 24.9212,C -2.0495,E1 25.1555,E2 76.7034} C_DIS
LIN {X 92.5205,Y 19.5855,Z 98,A 6.7518,B 24.9214,C -2.0476,E1 25.1565,E2 78.4476} C_DIS
LIN {X 93.0461,Y 16.9043,Z 98,A 5.108,B 24.9217,C -2.0429,E1 25.1574,E2 80.0929} C_DIS
LIN {X 93.4852,Y 14.2775,Z 98,A 3.4426,B 24.9223,C -2.0358,E1 25.1581,E2 81.765} C_DIS
LIN {X 93.8601,Y 11.5724,Z 98,A 1.8624,B 24.9225,C -2.0334,E1 25.1587,E2 83.3417} C_DIS
LIN {X 94.1535,Y 8.8572,Z 98,A 0.1267,B 24.9231,C -2.0251,E1 25.1592,E2 85.0867} C_DIS
LIN {X 94.3924,Y 5.8063,Z 98,A -1.6239,B 24.9233,C -2.0231,E1 25.1595,E2 86.8317} C_DIS
LIN {X 94.5255,Y 2.8706,Z 98,A -3.4939,B 24.9239,C -2.014,E1 25.1597,E2 88.712} C_DIS
LIN {X 94.5686,Y -0.309,Z 98,A -5.3305,B 24.9242,C -2.0112,E1 25.1597,E2 90.5443} C_DIS
LIN {X 94.5195,Y -3.0635,Z 98,A -7.0241,B 24.9246,C -2.0049,E1 25.1597,E2 92.2427} C_DIS
LIN {X 94.355,Y -6.3591,Z 98,A -9.0651,B 24.9252,C -1.9969,E1 25.1593,E2 94.2905} C_DIS
LIN {X 94.0717,Y -9.6871,Z 98,A -11.0662,B 24.9257,C -1.9912,E1 25.1588,E2 96.2931} C_DIS
LIN {X 93.7106,Y -12.7261,Z 98,A -12.9666,B 24.9262,C -1.9834,E1 25.1581,E2 98.2006} C_DIS
LIN {X 93.2482,Y -15.7512,Z 98,A -14.7006,B 24.9263,C -1.9821,E1 25.1574,E2 99.9277} C_DIS
LIN {X 92.7561,Y -18.4373,Z 98,A -16.2838,B 24.9265,C -1.9794,E1 25.1565,E2 101.5078} C_DIS
LIN {X 92.1761,Y -21.14,Z 98,A -18.0322,B 24.9271,C -1.9713,E1 25.1555,E2 103.2652} C_DIS
LIN {X 91.4478,Y -24.1027,Z 98,A -19.7806,B 24.9273,C -1.9692,E1 25.1543,E2 105.0084} C_DIS
LIN {X 90.6524,Y -26.9341,Z 98,A -21.6645,B 24.928,C -1.9598,E1 25.1528,E2 106.9039} C_DIS
LIN {X 89.7889,Y -29.691,Z 98,A -23.4512,B 24.9285,C -1.9529,E1 25.1513,E2 108.6966} C_DIS
LIN {X 88.8116,Y -32.4934,Z 98,A -25.1538,B 24.9286,C -1.9509,E1 25.1497,E2 110.3944} C_DIS
LIN {X 87.647,Y -35.5152,Z 98,A -27.1121,B 24.9291,C -1.9451,E1 25.1477,E2 112.3557} C_DIS
LIN {X 86.4554,Y -38.3287,Z 98,A -29.0322,B 24.9297,C -1.9368,E1 25.1455,E2 114.2848} C_DIS
LIN {X 85.1683,Y -41.1059,Z 98,A -30.7822,B 24.9297,C -1.9352,E1 25.1435,E2 116.0291} C_DIS
LIN {X 83.7399,Y -43.9426,Z 98,A -32.7048,B 24.9302,C -1.9295,E1 25.141,E2 117.9548} C_DIS
LIN {X 82.2787,Y -46.6246,Z 98,A -34.4537,B 24.9303,C -1.9279,E1 25.1386,E2 119.6984} C_DIS
LIN {X 81.1138,Y -48.6229,Z 98,A -36.0165,B 24.931,C -1.9178,E1 25.1364,E2 121.277} C_DIS
LIN {X 79.4108,Y -51.3549,Z 98,A -38.0139,B 24.9316,C -1.9105,E1 25.1334,E2 123.2816} C_DIS
LIN {X 77.5193,Y -54.1675,Z 98,A -40.0567,B 24.9319,C -1.9052,E1 25.1302,E2 125.3268} C_DIS
LIN {X 75.4998,Y -56.9484,Z 98,A -42.1106,B 24.9323,C -1.9006,E1 25.1267,E2 127.3818} C_DIS
LIN {X 73.3467,Y -59.696,Z 98,A -44.2005,B 24.9326,C -1.896,E1 25.1231,E2 129.4729} C_DIS
LIN {X 70.7411,Y -62.7629,Z 98,A -46.6123,B 24.933,C -1.8906,E1 25.1187,E2 131.8864} C_DIS
LIN {X 68.2989,Y -65.4114,Z 98,A -48.7486,B 24.9333,C -1.8869,E1 25.1146,E2 134.0222} C_DIS
LIN {X 65.7364,Y -67.9856,Z 98,A -50.9072,B 24.9335,C -1.8832,E1 25.1103,E2 136.1806} C_DIS
LIN {X 63.2917,Y -70.2677,Z 98,A -52.9108,B 24.9338,C -1.8792,E1 25.1062,E2 138.1853} C_DIS
LIN {X 60.8599,Y -72.3855,Z 98,A -54.9486,B 24.9343,C -1.8717,E1 25.1018,E2 140.233} C_DIS
LIN {X 58.1865,Y -74.5518,Z 98,A -57.0023,B 24.9346,C -1.8683,E1 25.0974,E2 142.2871} C_DIS
LIN {X 55.7097,Y -76.4184,Z 98,A -58.7559,B 24.9346,C -1.869,E1 25.0934,E2 144.0328} C_DIS
LIN {X 53.487,Y -77.992,Z 98,A -60.4995,B 24.935,C -1.8622,E1 25.0894,E2 145.7865} C_DIS
LIN {X 51.2163,Y -79.4998,Z 98,A -62.0678,B 24.935,C -1.862,E1 25.0858,E2 147.35} C_DIS
LIN {X 48.6227,Y -81.1139,Z 98,A -63.9887,B 24.9354,C -1.856,E1 25.0812,E2 149.2792} C_DIS
LIN {X 46.2407,Y -82.4932,Z 98,A -65.4816,B 24.9352,C -1.8594,E1 25.0776,E2 150.7595} C_DIS
LIN {X 43.9149,Y -83.7545,Z 98,A -67.1406,B 24.9355,C -1.8546,E1 25.0735,E2 152.4252} C_DIS
LIN {X 40.9135,Y -85.2607,Z 98,A -69.2551,B 24.936,C -1.8484,E1 25.0682,E2 154.5487} C_DIS
LIN {X 37.8676,Y -86.6565,Z 98,A -71.1231,B 24.9358,C -1.8511,E1 25.0634,E2 156.4055} C_DIS
LIN {X 35.7659,Y -87.545,Z 98,A -72.6072,B 24.9362,C -1.8455,E1 25.0596,E2 157.8997} C_DIS
LIN {X 32.9448,Y -88.6469,Z 98,A -74.3343,B 24.9361,C -1.8468,E1 25.0551,E2 159.6197} C_DIS
LIN {X 30.3958,Y -89.5513,Z 98,A -76.0625,B 24.9364,C -1.8415,E1 25.0505,E2 161.3571} C_DIS
LIN {X 27.4449,Y -90.5009,Z 98,A -78.0138,B 24.9368,C -1.8367,E1 25.0453,E2 163.3163} C_DIS
LIN {X 24.5014,Y -91.3401,Z 98,A -79.7555,B 24.9366,C -1.8387,E1 25.0406,E2 165.0503} C_DIS
LIN {X 21.8535,Y -92.0112,Z 98,A -81.5194,B 24.937,C -1.8332,E1 25.0358,E2 166.8247} C_DIS
LIN {X 19.1626,Y -92.6073,Z 98,A -83.1021,B 24.9369,C -1.8348,E1 25.0315,E2 168.4016} C_DIS
LIN {X 16.1578,Y -93.1802,Z 98,A -84.8604,B 24.9368,C -1.8366,E1 25.0267,E2 170.1535} C_DIS
LIN {X 13.4607,Y -93.6063,Z 98,A -86.6058,B 24.9371,C -1.8323,E1 25.0218,E2 171.9077} C_DIS
LIN {X 10.394,Y -93.9977,Z 98,A -88.5503,B 24.9373,C -1.8286,E1 25.0164,E2 173.8595} C_DIS
LIN {X 7.3523,Y -94.283,Z 98,A -90.298,B 24.9371,C -1.8313,E1 25.0116,E2 175.5998} C_DIS
LIN {X 4.6306,Y -94.4573,Z 98,A -92.0535,B 24.9374,C -1.827,E1 25.0067,E2 177.3648} C_DIS
LIN {X 1.575,Y -94.5561,Z 98,A -93.7971,B 24.9372,C -1.8302,E1 25.0018,E2 179.1004} C_DIS
LIN {X 1.575,Y -94.5561,Z 98,A -93.7971,B 24.9372,C -1.8302,E1 25.0018,E2 179.1004} C_DIS
Enddeposition()
LIN {X 0.7009,Y -101.7664,Z 99,A -93.7509,B 24.9437,C -1.7327,E1 25.0013,E2 179.2856} C_DIS
Startdeposition()
$VEL.CP = VEL_PRINT
LIN {X -2.2229,Y -101.7451,Z 99,A -95.7052,B 24.9445,C -1.7206,E1 24.9958,E2 181.2685} C_DIS
Enddeposition()
END
